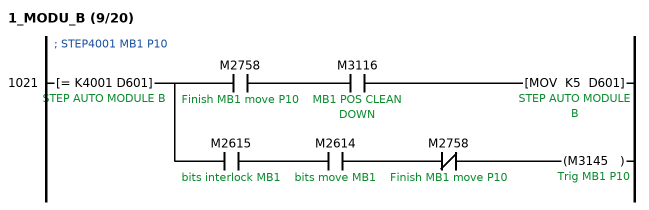
[picture p24: ladder of 1_MODU_B, rungs at steps 1021 to 1021]
; STEP4001 MB1 P10
1021  LD=     K4001 D601  ; STEP AUTO MODULE B
      MPS
      AND     M2758  ; Finish MB1 move P10
      AND     M3116  ; MB1 POS CLEAN DOWN
      MOV     K5 D601
      MPP
      AND     M2615  ; bits interlock MB1
      AND     M2614  ; bits move MB1
      ANI     M2758  ; Finish MB1 move P10
      OUT     M3145  ; Trig MB1 P10
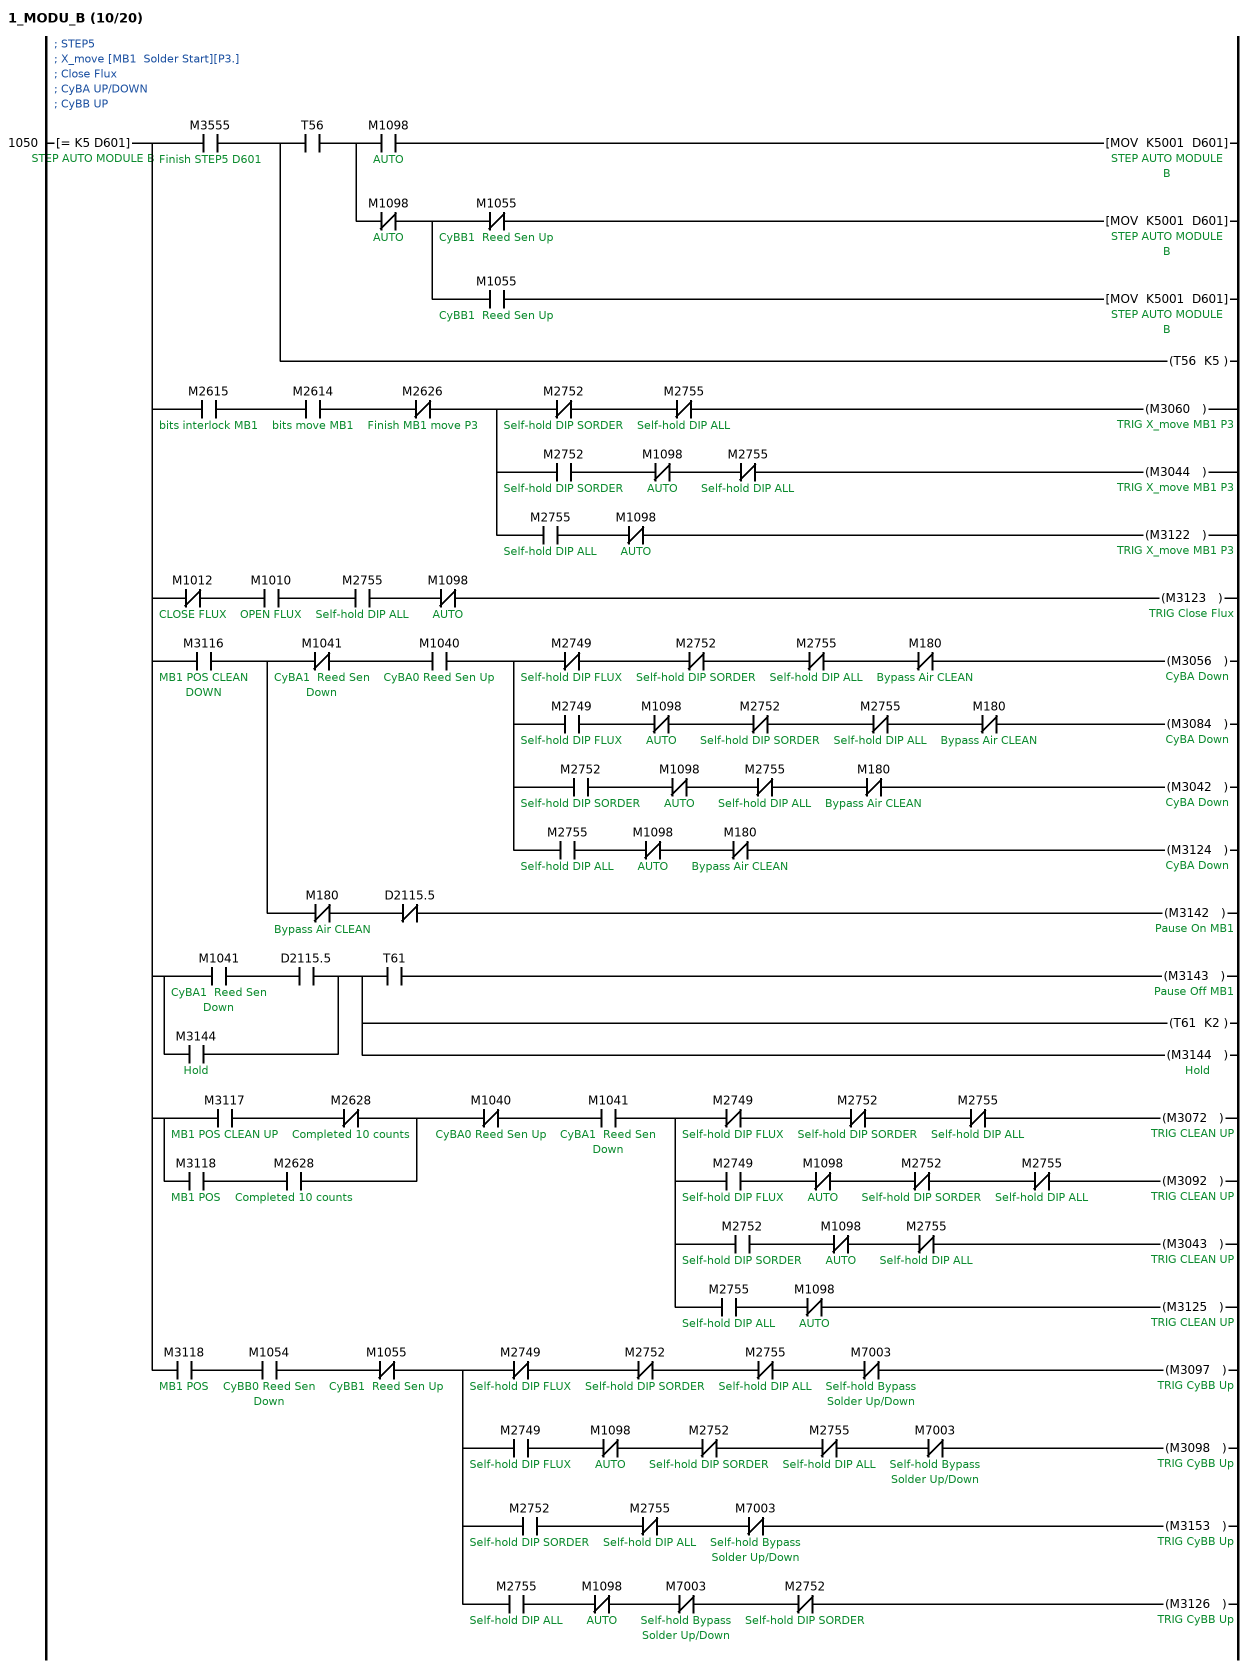
; STEP5
; X_move [MB1  Solder Start][P3.]
; Close Flux
; CyBA UP/DOWN
; CyBB UP
1050  LD=     K5 D601  ; STEP AUTO MODULE B
      MPS
      AND     M3555  ; Finish STEP5 D601
      MPS
      AND     T56
      MPS
      AND     M1098  ; AUTO
      MOV     K5001 D601
      MPP
      ANI     M1098  ; AUTO
      MPS
      ANI     M1055  ; CyBB1  Reed Sen Up
      MOV     K5001 D601
      MPP
      AND     M1055  ; CyBB1  Reed Sen Up
      MOV     K5001 D601
      MPP
      OUT     T56 K5
      MRD
      AND     M2615  ; bits interlock MB1
      AND     M2614  ; bits move MB1
      ANI     M2626  ; Finish MB1 move P3
      MPS
      ANI     M2752  ; Self-hold DIP SORDER
      ANI     M2755  ; Self-hold DIP ALL
      OUT     M3060  ; TRIG X_move MB1 P3
        [note] TRIG X_move MB1 P3
      MRD
      AND     M2752  ; Self-hold DIP SORDER
      ANI     M1098  ; AUTO
      ANI     M2755  ; Self-hold DIP ALL
      OUT     M3044  ; TRIG X_move MB1 P3
      MPP
      AND     M2755  ; Self-hold DIP ALL
      ANI     M1098  ; AUTO
      OUT     M3122  ; TRIG X_move MB1 P3
      MRD
      ANI     M1012  ; CLOSE FLUX
      AND     M1010  ; OPEN FLUX
      AND     M2755  ; Self-hold DIP ALL
      ANI     M1098  ; AUTO
      OUT     M3123  ; TRIG Close Flux
      MRD
      AND     M3116  ; MB1 POS CLEAN DOWN
      MPS
      ANI     M1041  ; CyBA1  Reed Sen Down
      AND     M1040  ; CyBA0 Reed Sen Up
      MPS
      ANI     M2749  ; Self-hold DIP FLUX
      ANI     M2752  ; Self-hold DIP SORDER
      ANI     M2755  ; Self-hold DIP ALL
      ANI     M180  ; Bypass Air CLEAN
      OUT     M3056  ; CyBA Down
        [note] TRIG CLEAN DOWN
      MRD
      AND     M2749  ; Self-hold DIP FLUX
      ANI     M1098  ; AUTO
      ANI     M2752  ; Self-hold DIP SORDER
      ANI     M2755  ; Self-hold DIP ALL
      ANI     M180  ; Bypass Air CLEAN
      OUT     M3084  ; CyBA Down
      MRD
      AND     M2752  ; Self-hold DIP SORDER
      ANI     M1098  ; AUTO
      ANI     M2755  ; Self-hold DIP ALL
      ANI     M180  ; Bypass Air CLEAN
      OUT     M3042  ; CyBA Down
      MPP
      AND     M2755  ; Self-hold DIP ALL
      ANI     M1098  ; AUTO
      ANI     M180  ; Bypass Air CLEAN
      OUT     M3124  ; CyBA Down
      MPP
      ANI     M180  ; Bypass Air CLEAN
      ANI     D2115.5
      OUT     M3142  ; Pause On MB1
      MRD
      LD      M1041  ; CyBA1  Reed Sen Down
      AND     D2115.5
      OR      M3144  ; Hold
      ANB
      MPS
      AND     T61
      OUT     M3143  ; Pause Off MB1
      MPP
      OUT     T61 K2
      OUT     M3144  ; Hold
      MRD
      LD      M3117  ; MB1 POS CLEAN UP
      ANI     M2628  ; Completed 10 counts
      LD      M3118  ; MB1 POS
      AND     M2628  ; Completed 10 counts
      ORB
      ANB
      ANI     M1040  ; CyBA0 Reed Sen Up
      AND     M1041  ; CyBA1  Reed Sen Down
      MPS
      ANI     M2749  ; Self-hold DIP FLUX
      ANI     M2752  ; Self-hold DIP SORDER
      ANI     M2755  ; Self-hold DIP ALL
      OUT     M3072  ; TRIG CLEAN UP
        [note] TRIG CLEAN UP
      MRD
      AND     M2749  ; Self-hold DIP FLUX
      ANI     M1098  ; AUTO
      ANI     M2752  ; Self-hold DIP SORDER
      ANI     M2755  ; Self-hold DIP ALL
      OUT     M3092  ; TRIG CLEAN UP
      MRD
      AND     M2752  ; Self-hold DIP SORDER
      ANI     M1098  ; AUTO
      ANI     M2755  ; Self-hold DIP ALL
      OUT     M3043  ; TRIG CLEAN UP
      MPP
      AND     M2755  ; Self-hold DIP ALL
      ANI     M1098  ; AUTO
      OUT     M3125  ; TRIG CLEAN UP
      MPP
      AND     M3118  ; MB1 POS
      AND     M1054  ; CyBB0 Reed Sen Down
      ANI     M1055  ; CyBB1  Reed Sen Up
      MPS
      ANI     M2749  ; Self-hold DIP FLUX
      ANI     M2752  ; Self-hold DIP SORDER
      ANI     M2755  ; Self-hold DIP ALL
      ANI     M7003  ; Self-hold Bypass Solder Up/Down
      OUT     M3097  ; TRIG CyBB Up
        [note] TRIG CyBB Up
      MRD
      AND     M2749  ; Self-hold DIP FLUX
      ANI     M1098  ; AUTO
      ANI     M2752  ; Self-hold DIP SORDER
      ANI     M2755  ; Self-hold DIP ALL
      ANI     M7003  ; Self-hold Bypass Solder Up/Down
      OUT     M3098  ; TRIG CyBB Up
      MRD
      AND     M2752  ; Self-hold DIP SORDER
      ANI     M2755  ; Self-hold DIP ALL
      ANI     M7003  ; Self-hold Bypass Solder Up/Down
      OUT     M3153  ; TRIG CyBB Up
      MPP
      AND     M2755  ; Self-hold DIP ALL
      ANI     M1098  ; AUTO
      ANI     M7003  ; Self-hold Bypass Solder Up/Down
      ANI     M2752  ; Self-hold DIP SORDER
      OUT     M3126  ; TRIG CyBB Up
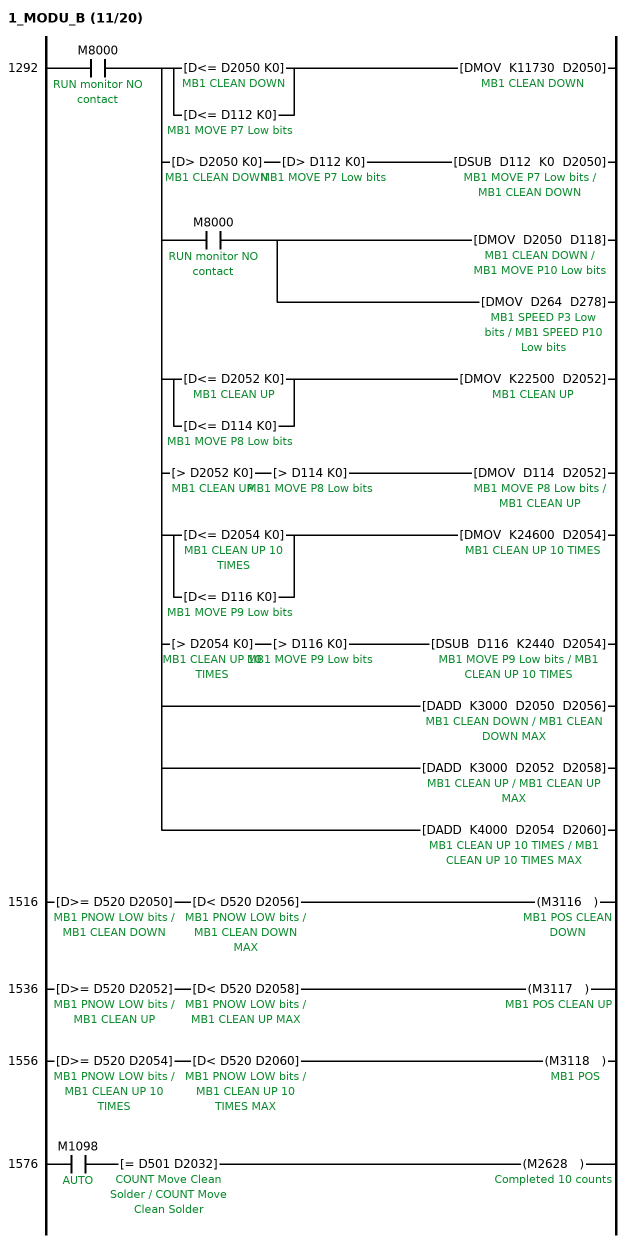
1292  LD      M8000  ; RUN monitor NO contact
      MPS
      LDD<=   D2050 K0  ; MB1 CLEAN DOWN
      ORD<=   D112 K0  ; MB1 MOVE P7 Low bits
      ANB
      DMOV    K11730 D2050
      MRD
      ANDD>   D2050 K0  ; MB1 CLEAN DOWN
      ANDD>   D112 K0  ; MB1 MOVE P7 Low bits
      DSUB    D112 K0 D2050
      MRD
      AND     M8000  ; RUN monitor NO contact
      DMOV    D2050 D118  ; MB1 MOVE P10 Low bits
      DMOV    D264 D278  ; MB1 SPEED P3 Low bits / MB1 SPEED P10 Low bits
      MRD
      LDD<=   D2052 K0  ; MB1 CLEAN UP
      ORD<=   D114 K0  ; MB1 MOVE P8 Low bits
      ANB
      DMOV    K22500 D2052
      MRD
      AND>    D2052 K0  ; MB1 CLEAN UP
      AND>    D114 K0  ; MB1 MOVE P8 Low bits
      DMOV    D114 D2052
      MRD
      LDD<=   D2054 K0  ; MB1 CLEAN UP 10 TIMES
      ORD<=   D116 K0  ; MB1 MOVE P9 Low bits
      ANB
      DMOV    K24600 D2054
      MRD
      AND>    D2054 K0  ; MB1 CLEAN UP 10 TIMES
      AND>    D116 K0  ; MB1 MOVE P9 Low bits
      DSUB    D116 K2440 D2054
      MPP
      DADD    K3000 D2050 D2056  ; MB1 CLEAN DOWN MAX
      DADD    K3000 D2052 D2058  ; MB1 CLEAN UP MAX
      DADD    K4000 D2054 D2060  ; MB1 CLEAN UP 10 TIMES MAX
1516  LDD>=   D520 D2050  ; MB1 PNOW LOW bits / MB1 CLEAN DOWN
      ANDD<   D520 D2056  ; MB1 PNOW LOW bits / MB1 CLEAN DOWN MAX
      OUT     M3116  ; MB1 POS CLEAN DOWN
1536  LDD>=   D520 D2052  ; MB1 PNOW LOW bits / MB1 CLEAN UP
      ANDD<   D520 D2058  ; MB1 PNOW LOW bits / MB1 CLEAN UP MAX
      OUT     M3117  ; MB1 POS CLEAN UP
1556  LDD>=   D520 D2054  ; MB1 PNOW LOW bits / MB1 CLEAN UP 10 TIMES
      ANDD<   D520 D2060  ; MB1 PNOW LOW bits / MB1 CLEAN UP 10 TIMES MAX
      OUT     M3118  ; MB1 POS
1576  LD      M1098  ; AUTO
      AND=    D501 D2032  ; COUNT Move Clean Solder / COUNT Move Clean Solder
      OUT     M2628  ; Completed 10 counts
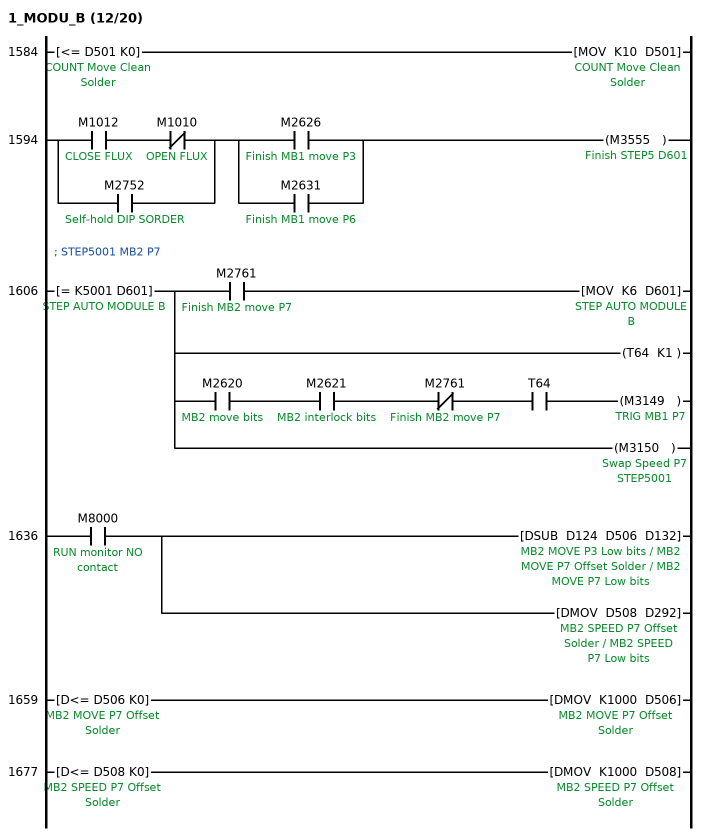
1584  LD<=    D501 K0  ; COUNT Move Clean Solder
      MOV     K10 D501
1594  LD      M1012  ; CLOSE FLUX
      ANI     M1010  ; OPEN FLUX
      OR      M2752  ; Self-hold DIP SORDER
      LD      M2626  ; Finish MB1 move P3
      OR      M2631  ; Finish MB1 move P6
      ANB
      OUT     M3555  ; Finish STEP5 D601
; STEP5001 MB2 P7
1606  LD=     K5001 D601  ; STEP AUTO MODULE B
      MPS
      AND     M2761  ; Finish MB2 move P7
      MOV     K6 D601
      MPP
      OUT     T64 K1
      MPS
      AND     M2620  ; MB2 move bits
      AND     M2621  ; MB2 interlock bits
      ANI     M2761  ; Finish MB2 move P7
      AND     T64
      OUT     M3149  ; TRIG MB1 P7
      MPP
      OUT     M3150  ; Swap Speed P7 STEP5001
1636  LD      M8000  ; RUN monitor NO contact
      DSUB    D124 D506 D132  ; MB2 MOVE P3 Low bits / MB2 MOVE P7 Offset Solder / MB2 MOVE P7 Low bits
      DMOV    D508 D292  ; MB2 SPEED P7 Offset Solder / MB2 SPEED P7 Low bits
1659  LDD<=   D506 K0  ; MB2 MOVE P7 Offset Solder
      DMOV    K1000 D506
1677  LDD<=   D508 K0  ; MB2 SPEED P7 Offset Solder
      DMOV    K1000 D508
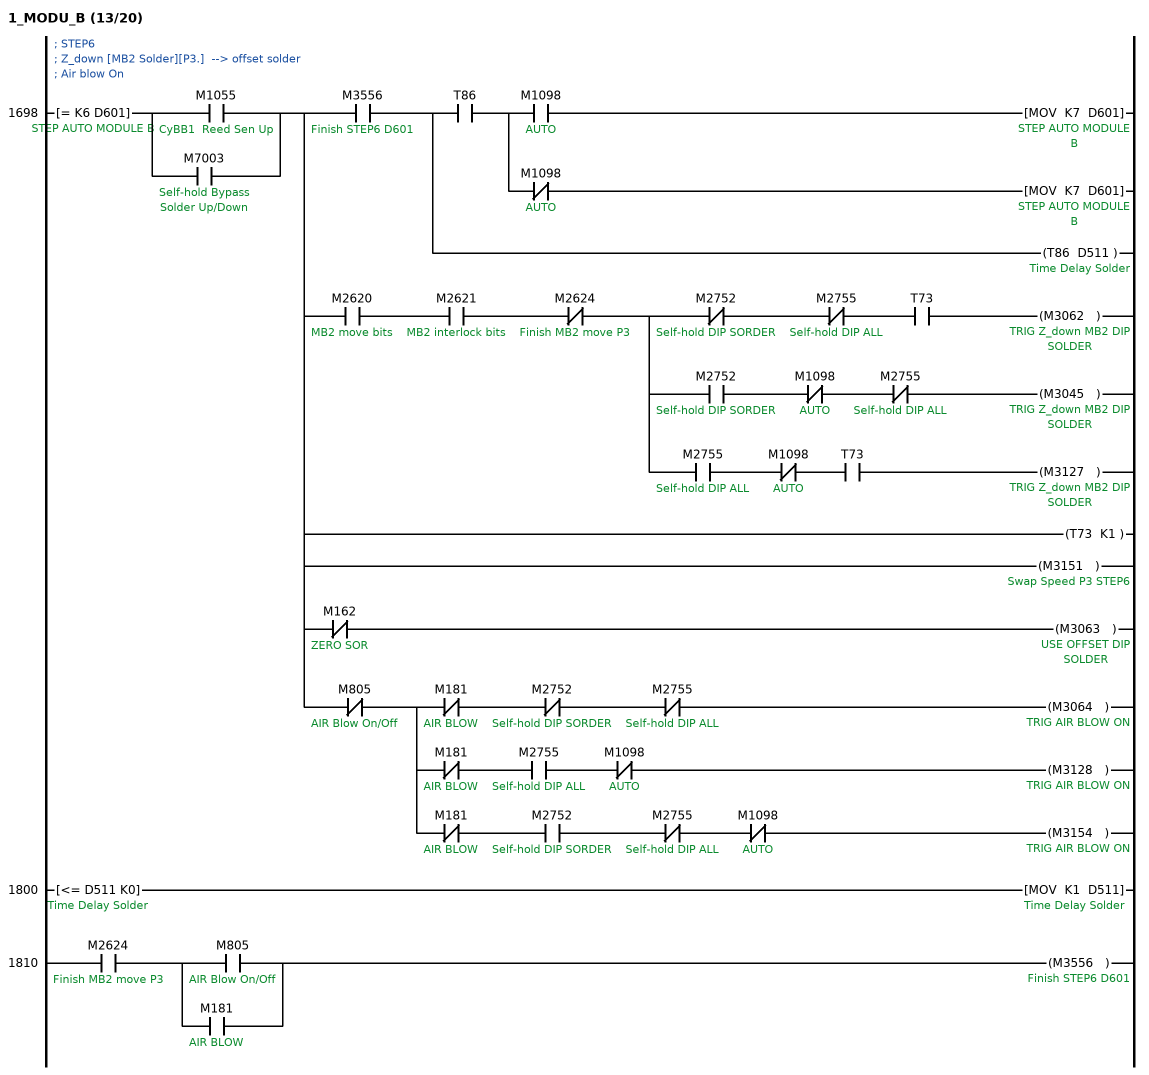
; STEP6
; Z_down [MB2 Solder][P3.]  --> offset solder
; Air blow On
1698  LD=     K6 D601  ; STEP AUTO MODULE B
      LD      M1055  ; CyBB1  Reed Sen Up
      OR      M7003  ; Self-hold Bypass Solder Up/Down
      ANB
      MPS
      AND     M3556  ; Finish STEP6 D601
      MPS
      AND     T86
      MPS
      AND     M1098  ; AUTO
      MOV     K7 D601
      MPP
      ANI     M1098  ; AUTO
      MOV     K7 D601
      MPP
      OUT     T86 D511  ; Time Delay Solder
      MRD
      AND     M2620  ; MB2 move bits
      AND     M2621  ; MB2 interlock bits
      ANI     M2624  ; Finish MB2 move P3
      MPS
      ANI     M2752  ; Self-hold DIP SORDER
      ANI     M2755  ; Self-hold DIP ALL
      AND     T73
      OUT     M3062  ; TRIG Z_down MB2 DIP SOLDER
        [note] TRIG Z_down MB2 DIP SOLDER
      MRD
      AND     M2752  ; Self-hold DIP SORDER
      ANI     M1098  ; AUTO
      ANI     M2755  ; Self-hold DIP ALL
      OUT     M3045  ; TRIG Z_down MB2 DIP SOLDER
      MPP
      AND     M2755  ; Self-hold DIP ALL
      ANI     M1098  ; AUTO
      AND     T73
      OUT     M3127  ; TRIG Z_down MB2 DIP SOLDER
      MPP
      OUT     T73 K1
      OUT     M3151  ; Swap Speed P3 STEP6
      MPS
      ANI     M162  ; ZERO SOR
      OUT     M3063  ; USE OFFSET DIP SOLDER
        [note] USE OFFSET DIP SOLDER
      MPP
      ANI     M805  ; AIR Blow On/Off
      MPS
      ANI     M181  ; AIR BLOW
      ANI     M2752  ; Self-hold DIP SORDER
      ANI     M2755  ; Self-hold DIP ALL
      OUT     M3064  ; TRIG AIR BLOW ON
        [note] TRIG AIR BLOW ON
      MRD
      ANI     M181  ; AIR BLOW
      AND     M2755  ; Self-hold DIP ALL
      ANI     M1098  ; AUTO
      OUT     M3128  ; TRIG AIR BLOW ON
      MPP
      ANI     M181  ; AIR BLOW
      AND     M2752  ; Self-hold DIP SORDER
      ANI     M2755  ; Self-hold DIP ALL
      ANI     M1098  ; AUTO
      OUT     M3154  ; TRIG AIR BLOW ON
1800  LD<=    D511 K0  ; Time Delay Solder
      MOV     K1 D511
1810  LD      M2624  ; Finish MB2 move P3
      LD      M805  ; AIR Blow On/Off
      OR      M181  ; AIR BLOW
      ANB
      OUT     M3556  ; Finish STEP6 D601
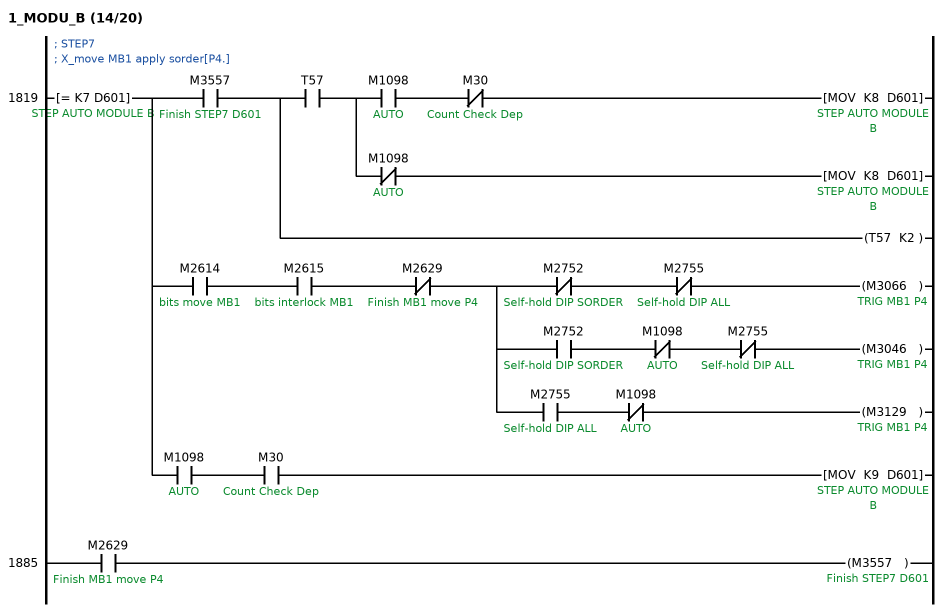
; STEP7
; X_move MB1 apply sorder[P4.]
1819  LD=     K7 D601  ; STEP AUTO MODULE B
      MPS
      AND     M3557  ; Finish STEP7 D601
      MPS
      AND     T57
      MPS
      AND     M1098  ; AUTO
      ANI     M30  ; Count Check Dep
      MOV     K8 D601
      MPP
      ANI     M1098  ; AUTO
      MOV     K8 D601
      MPP
      OUT     T57 K2
      MRD
      AND     M2614  ; bits move MB1
      AND     M2615  ; bits interlock MB1
      ANI     M2629  ; Finish MB1 move P4
      MPS
      ANI     M2752  ; Self-hold DIP SORDER
      ANI     M2755  ; Self-hold DIP ALL
      OUT     M3066  ; TRIG MB1 P4
        [note] TRIG MB1 P4
      MRD
      AND     M2752  ; Self-hold DIP SORDER
      ANI     M1098  ; AUTO
      ANI     M2755  ; Self-hold DIP ALL
      OUT     M3046  ; TRIG MB1 P4
      MPP
      AND     M2755  ; Self-hold DIP ALL
      ANI     M1098  ; AUTO
      OUT     M3129  ; TRIG MB1 P4
      MPP
      AND     M1098  ; AUTO
      AND     M30  ; Count Check Dep
      MOV     K9 D601
1885  LD      M2629  ; Finish MB1 move P4
      OUT     M3557  ; Finish STEP7 D601
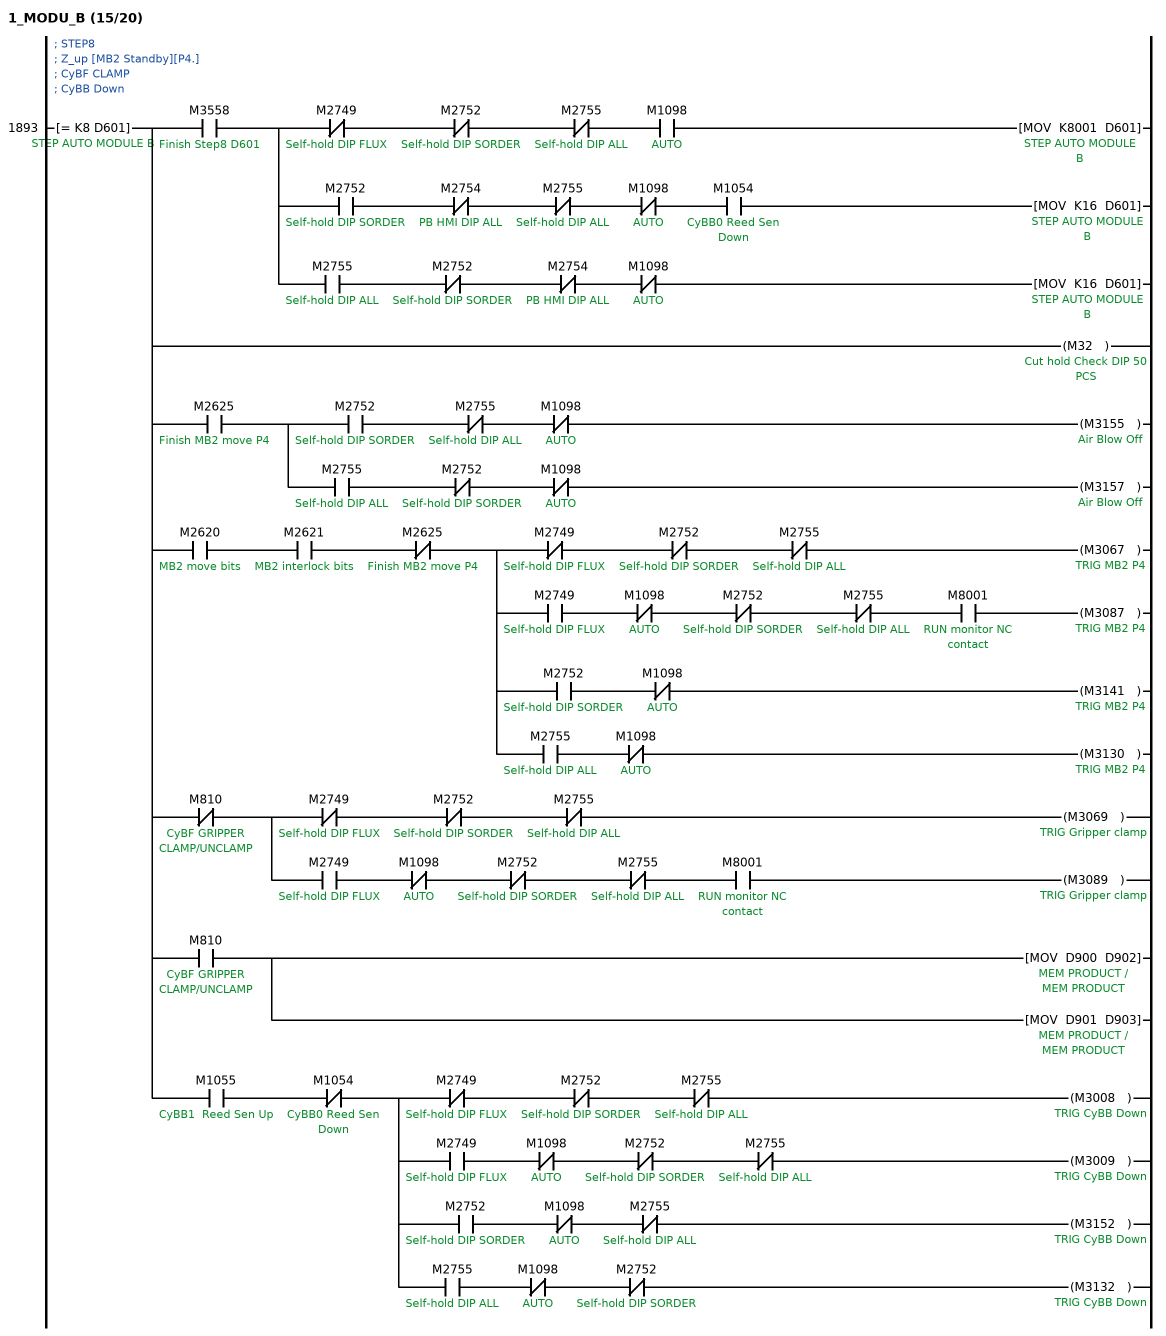
; STEP8
; Z_up [MB2 Standby][P4.]
; CyBF CLAMP
; CyBB Down
1893  LD=     K8 D601  ; STEP AUTO MODULE B
      MPS
      AND     M3558  ; Finish Step8 D601
      MPS
      ANI     M2749  ; Self-hold DIP FLUX
      ANI     M2752  ; Self-hold DIP SORDER
      ANI     M2755  ; Self-hold DIP ALL
      AND     M1098  ; AUTO
      MOV     K8001 D601
      MRD
      AND     M2752  ; Self-hold DIP SORDER
      ANI     M2754  ; PB HMI DIP ALL
      ANI     M2755  ; Self-hold DIP ALL
      ANI     M1098  ; AUTO
      AND     M1054  ; CyBB0 Reed Sen Down
      MOV     K16 D601
      MPP
      AND     M2755  ; Self-hold DIP ALL
      ANI     M2752  ; Self-hold DIP SORDER
      ANI     M2754  ; PB HMI DIP ALL
      ANI     M1098  ; AUTO
      MOV     K16 D601
      MPP
      OUT     M32  ; Cut hold Check DIP 50 PCS
      MPS
      AND     M2625  ; Finish MB2 move P4
      MPS
      AND     M2752  ; Self-hold DIP SORDER
      ANI     M2755  ; Self-hold DIP ALL
      ANI     M1098  ; AUTO
      OUT     M3155  ; Air Blow Off
      MPP
      AND     M2755  ; Self-hold DIP ALL
      ANI     M2752  ; Self-hold DIP SORDER
      ANI     M1098  ; AUTO
      OUT     M3157  ; Air Blow Off
      MRD
      AND     M2620  ; MB2 move bits
      AND     M2621  ; MB2 interlock bits
      ANI     M2625  ; Finish MB2 move P4
      MPS
      ANI     M2749  ; Self-hold DIP FLUX
      ANI     M2752  ; Self-hold DIP SORDER
      ANI     M2755  ; Self-hold DIP ALL
      OUT     M3067  ; TRIG MB2 P4
        [note] TRIG MB2 P4
      MRD
      AND     M2749  ; Self-hold DIP FLUX
      ANI     M1098  ; AUTO
      ANI     M2752  ; Self-hold DIP SORDER
      ANI     M2755  ; Self-hold DIP ALL
      AND     M8001  ; RUN monitor NC contact
      OUT     M3087  ; TRIG MB2 P4
      MRD
      AND     M2752  ; Self-hold DIP SORDER
      ANI     M1098  ; AUTO
      OUT     M3141  ; TRIG MB2 P4
      MPP
      AND     M2755  ; Self-hold DIP ALL
      ANI     M1098  ; AUTO
      OUT     M3130  ; TRIG MB2 P4
      MRD
      ANI     M810  ; CyBF GRIPPER CLAMP/UNCLAMP
      MPS
      ANI     M2749  ; Self-hold DIP FLUX
      ANI     M2752  ; Self-hold DIP SORDER
      ANI     M2755  ; Self-hold DIP ALL
      OUT     M3069  ; TRIG Gripper clamp
        [note] TRIG Gripper clamp
      MPP
      AND     M2749  ; Self-hold DIP FLUX
      ANI     M1098  ; AUTO
      ANI     M2752  ; Self-hold DIP SORDER
      ANI     M2755  ; Self-hold DIP ALL
      AND     M8001  ; RUN monitor NC contact
      OUT     M3089  ; TRIG Gripper clamp
      MRD
      AND     M810  ; CyBF GRIPPER CLAMP/UNCLAMP
      MOV     D900 D902
      MOV     D901 D903
      MPP
      AND     M1055  ; CyBB1  Reed Sen Up
      ANI     M1054  ; CyBB0 Reed Sen Down
      MPS
      ANI     M2749  ; Self-hold DIP FLUX
      ANI     M2752  ; Self-hold DIP SORDER
      ANI     M2755  ; Self-hold DIP ALL
      OUT     M3008  ; TRIG CyBB Down
        [note] TRIG CyBB Down
      MRD
      AND     M2749  ; Self-hold DIP FLUX
      ANI     M1098  ; AUTO
      ANI     M2752  ; Self-hold DIP SORDER
      ANI     M2755  ; Self-hold DIP ALL
      OUT     M3009  ; TRIG CyBB Down
      MRD
      AND     M2752  ; Self-hold DIP SORDER
      ANI     M1098  ; AUTO
      ANI     M2755  ; Self-hold DIP ALL
      OUT     M3152  ; TRIG CyBB Down
      MPP
      AND     M2755  ; Self-hold DIP ALL
      ANI     M1098  ; AUTO
      ANI     M2752  ; Self-hold DIP SORDER
      OUT     M3132  ; TRIG CyBB Down
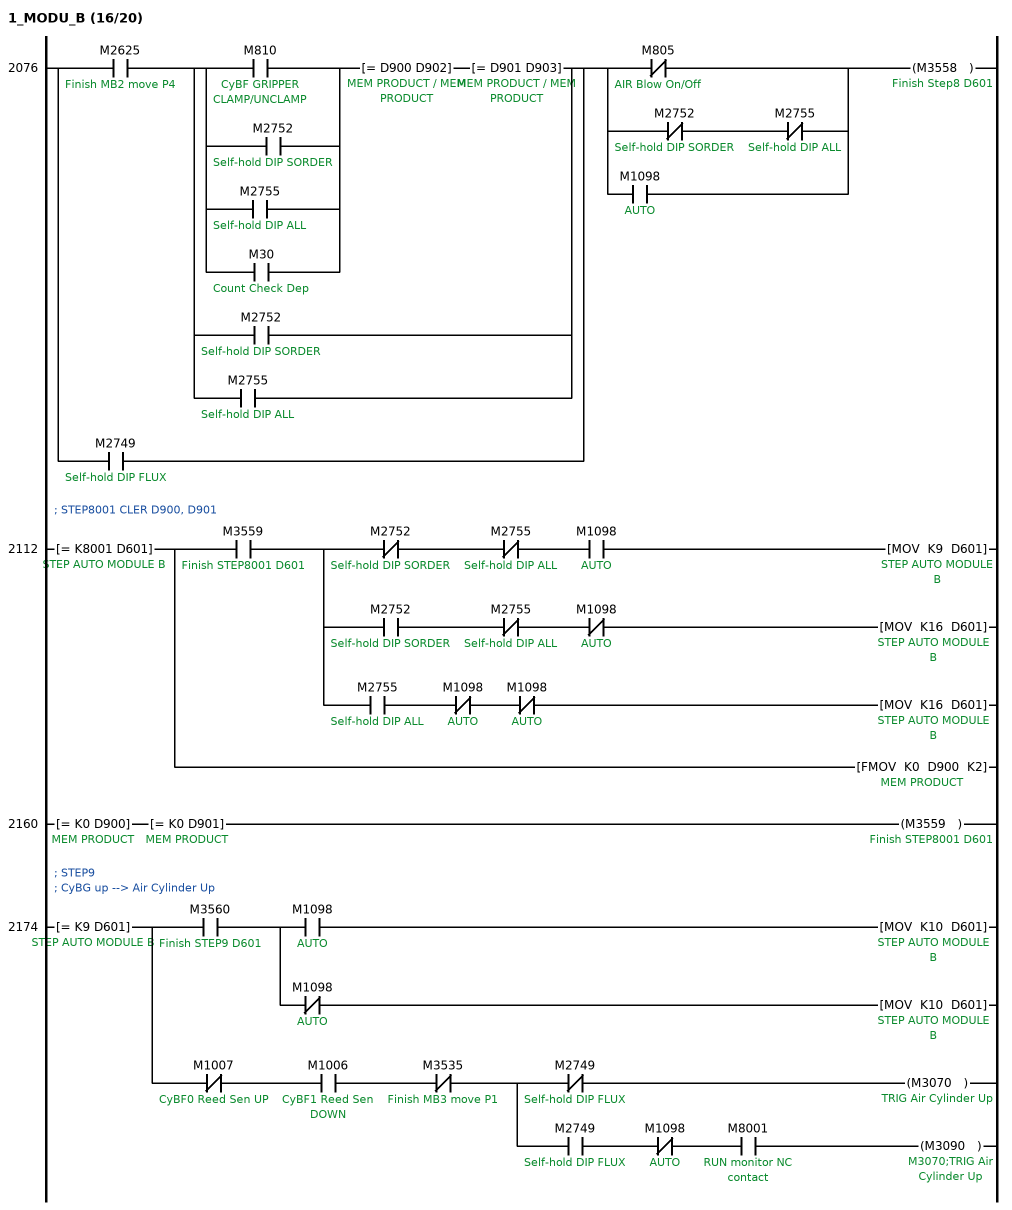
2076  LD      M2625  ; Finish MB2 move P4
      LD      M810  ; CyBF GRIPPER CLAMP/UNCLAMP
      OR      M2752  ; Self-hold DIP SORDER
      OR      M2755  ; Self-hold DIP ALL
      OR      M30  ; Count Check Dep
      AND=    D900 D902  ; MEM PRODUCT / MEM PRODUCT
      AND=    D901 D903  ; MEM PRODUCT / MEM PRODUCT
      OR      M2752  ; Self-hold DIP SORDER
      OR      M2755  ; Self-hold DIP ALL
      ANB
      OR      M2749  ; Self-hold DIP FLUX
      LDI     M805  ; AIR Blow On/Off
      LDI     M2752  ; Self-hold DIP SORDER
      ANI     M2755  ; Self-hold DIP ALL
      ORB
      OR      M1098  ; AUTO
      ANB
      OUT     M3558  ; Finish Step8 D601
; STEP8001 CLER D900, D901
2112  LD=     K8001 D601  ; STEP AUTO MODULE B
      MPS
      AND     M3559  ; Finish STEP8001 D601
      MPS
      ANI     M2752  ; Self-hold DIP SORDER
      ANI     M2755  ; Self-hold DIP ALL
      AND     M1098  ; AUTO
      MOV     K9 D601
      MRD
      AND     M2752  ; Self-hold DIP SORDER
      ANI     M2755  ; Self-hold DIP ALL
      ANI     M1098  ; AUTO
      MOV     K16 D601
      MPP
      AND     M2755  ; Self-hold DIP ALL
      ANI     M1098  ; AUTO
      ANI     M1098  ; AUTO
      MOV     K16 D601
      MPP
      FMOV    K0 D900 K2
2160  LD=     K0 D900  ; MEM PRODUCT
      AND=    K0 D901  ; MEM PRODUCT
      OUT     M3559  ; Finish STEP8001 D601
; STEP9
; CyBG up --> Air Cylinder Up
2174  LD=     K9 D601  ; STEP AUTO MODULE B
      MPS
      AND     M3560  ; Finish STEP9 D601
      MPS
      AND     M1098  ; AUTO
      MOV     K10 D601
      MPP
      ANI     M1098  ; AUTO
      MOV     K10 D601
      MPP
      ANI     M1007  ; CyBF0 Reed Sen UP
      AND     M1006  ; CyBF1 Reed Sen DOWN
      ANI     M3535  ; Finish MB3 move P1
      MPS
      ANI     M2749  ; Self-hold DIP FLUX
      OUT     M3070  ; TRIG Air Cylinder Up
        [note] TRIG Air Cylinder Up
      MPP
      AND     M2749  ; Self-hold DIP FLUX
      ANI     M1098  ; AUTO
      AND     M8001  ; RUN monitor NC contact
      OUT     M3090  ; M3070;TRIG Air Cylinder Up
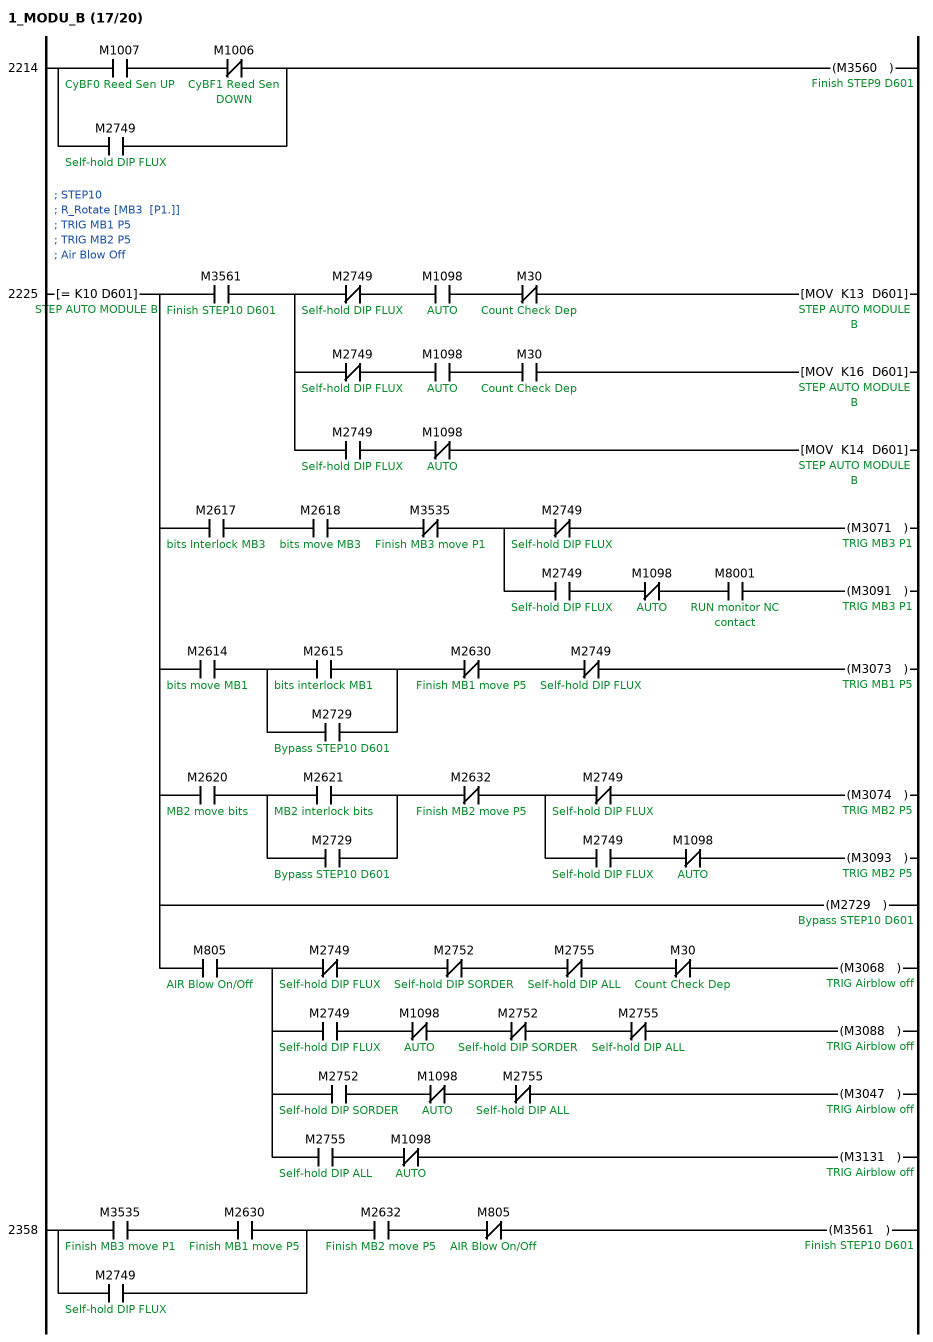
2214  LD      M1007  ; CyBF0 Reed Sen UP
      ANI     M1006  ; CyBF1 Reed Sen DOWN
      OR      M2749  ; Self-hold DIP FLUX
      OUT     M3560  ; Finish STEP9 D601
; STEP10
; R_Rotate [MB3  [P1.]]
; TRIG MB1 P5
; TRIG MB2 P5
; Air Blow Off
2225  LD=     K10 D601  ; STEP AUTO MODULE B
      MPS
      AND     M3561  ; Finish STEP10 D601
      MPS
      ANI     M2749  ; Self-hold DIP FLUX
      AND     M1098  ; AUTO
      ANI     M30  ; Count Check Dep
      MOV     K13 D601
      MRD
      ANI     M2749  ; Self-hold DIP FLUX
      AND     M1098  ; AUTO
      AND     M30  ; Count Check Dep
      MOV     K16 D601
      MPP
      AND     M2749  ; Self-hold DIP FLUX
      ANI     M1098  ; AUTO
      MOV     K14 D601
      MRD
      AND     M2617  ; bits Interlock MB3
      AND     M2618  ; bits move MB3
      ANI     M3535  ; Finish MB3 move P1
      MPS
      ANI     M2749  ; Self-hold DIP FLUX
      OUT     M3071  ; TRIG MB3 P1
        [note] TRIG MB3 P1
      MPP
      AND     M2749  ; Self-hold DIP FLUX
      ANI     M1098  ; AUTO
      AND     M8001  ; RUN monitor NC contact
      OUT     M3091  ; TRIG MB3 P1
      MRD
      AND     M2614  ; bits move MB1
      LD      M2615  ; bits interlock MB1
      OR      M2729  ; Bypass STEP10 D601
      ANB
      ANI     M2630  ; Finish MB1 move P5
      ANI     M2749  ; Self-hold DIP FLUX
      OUT     M3073  ; TRIG MB1 P5
        [note] TRIG MB1 P5
      MRD
      AND     M2620  ; MB2 move bits
      LD      M2621  ; MB2 interlock bits
      OR      M2729  ; Bypass STEP10 D601
      ANB
      ANI     M2632  ; Finish MB2 move P5
      MPS
      ANI     M2749  ; Self-hold DIP FLUX
      OUT     M3074  ; TRIG MB2 P5
        [note] TRIG MB2 P5
      MPP
      AND     M2749  ; Self-hold DIP FLUX
      ANI     M1098  ; AUTO
      OUT     M3093  ; TRIG MB2 P5
      MPP
      OUT     M2729  ; Bypass STEP10 D601
      AND     M805  ; AIR Blow On/Off
      MPS
      ANI     M2749  ; Self-hold DIP FLUX
      ANI     M2752  ; Self-hold DIP SORDER
      ANI     M2755  ; Self-hold DIP ALL
      ANI     M30  ; Count Check Dep
      OUT     M3068  ; TRIG Airblow off
        [note] TRIG Airblow off
      MRD
      AND     M2749  ; Self-hold DIP FLUX
      ANI     M1098  ; AUTO
      ANI     M2752  ; Self-hold DIP SORDER
      ANI     M2755  ; Self-hold DIP ALL
      OUT     M3088  ; TRIG Airblow off
      MRD
      AND     M2752  ; Self-hold DIP SORDER
      ANI     M1098  ; AUTO
      ANI     M2755  ; Self-hold DIP ALL
      OUT     M3047  ; TRIG Airblow off
      MPP
      AND     M2755  ; Self-hold DIP ALL
      ANI     M1098  ; AUTO
      OUT     M3131  ; TRIG Airblow off
2358  LD      M3535  ; Finish MB3 move P1
      AND     M2630  ; Finish MB1 move P5
      OR      M2749  ; Self-hold DIP FLUX
      AND     M2632  ; Finish MB2 move P5
      ANI     M805  ; AIR Blow On/Off
      OUT     M3561  ; Finish STEP10 D601
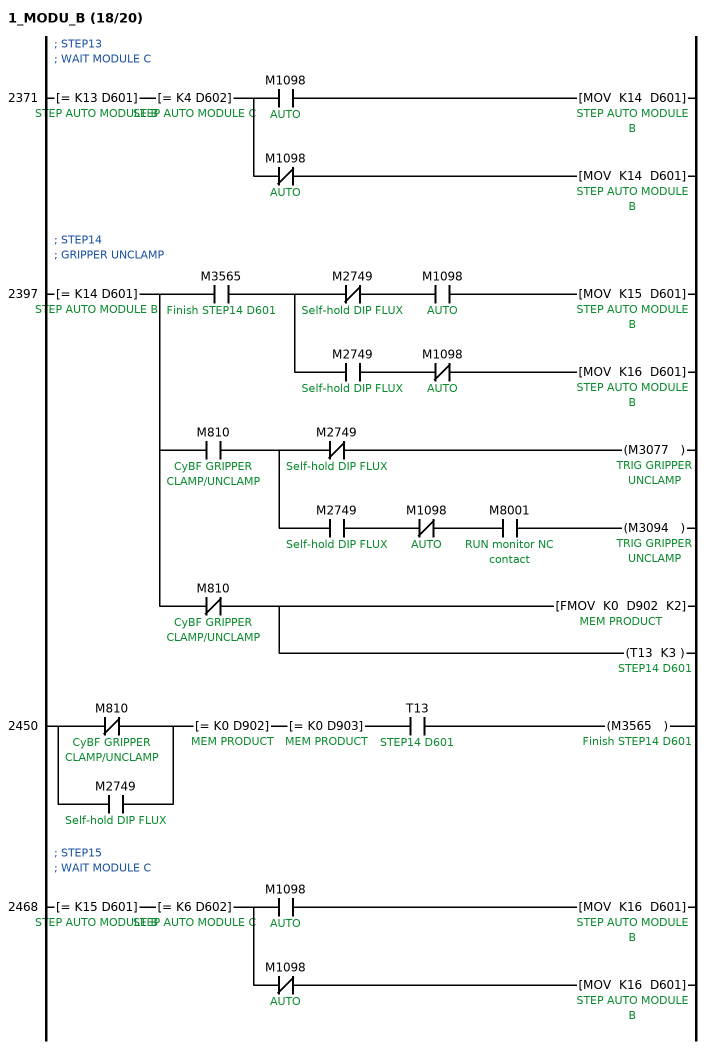
; STEP13
; WAIT MODULE C
2371  LD=     K13 D601  ; STEP AUTO MODULE B
      AND=    K4 D602  ; STEP AUTO MODULE C
      MPS
      AND     M1098  ; AUTO
      MOV     K14 D601
      MPP
      ANI     M1098  ; AUTO
      MOV     K14 D601
; STEP14
; GRIPPER UNCLAMP
2397  LD=     K14 D601  ; STEP AUTO MODULE B
      MPS
      AND     M3565  ; Finish STEP14 D601
      MPS
      ANI     M2749  ; Self-hold DIP FLUX
      AND     M1098  ; AUTO
      MOV     K15 D601
      MPP
      AND     M2749  ; Self-hold DIP FLUX
      ANI     M1098  ; AUTO
      MOV     K16 D601
      MRD
      AND     M810  ; CyBF GRIPPER CLAMP/UNCLAMP
      MPS
      ANI     M2749  ; Self-hold DIP FLUX
      OUT     M3077  ; TRIG GRIPPER UNCLAMP
        [note] TRIG GRIPPER UNCLAMP
      MPP
      AND     M2749  ; Self-hold DIP FLUX
      ANI     M1098  ; AUTO
      AND     M8001  ; RUN monitor NC contact
      OUT     M3094  ; TRIG GRIPPER UNCLAMP
      MPP
      ANI     M810  ; CyBF GRIPPER CLAMP/UNCLAMP
      FMOV    K0 D902 K2
      OUT     T13 K3  ; STEP14 D601
2450  LDI     M810  ; CyBF GRIPPER CLAMP/UNCLAMP
      OR      M2749  ; Self-hold DIP FLUX
      AND=    K0 D902  ; MEM PRODUCT
      AND=    K0 D903  ; MEM PRODUCT
      AND     T13  ; STEP14 D601
      OUT     M3565  ; Finish STEP14 D601
; STEP15
; WAIT MODULE C
2468  LD=     K15 D601  ; STEP AUTO MODULE B
      AND=    K6 D602  ; STEP AUTO MODULE C
      MPS
      AND     M1098  ; AUTO
      MOV     K16 D601
      MPP
      ANI     M1098  ; AUTO
      MOV     K16 D601
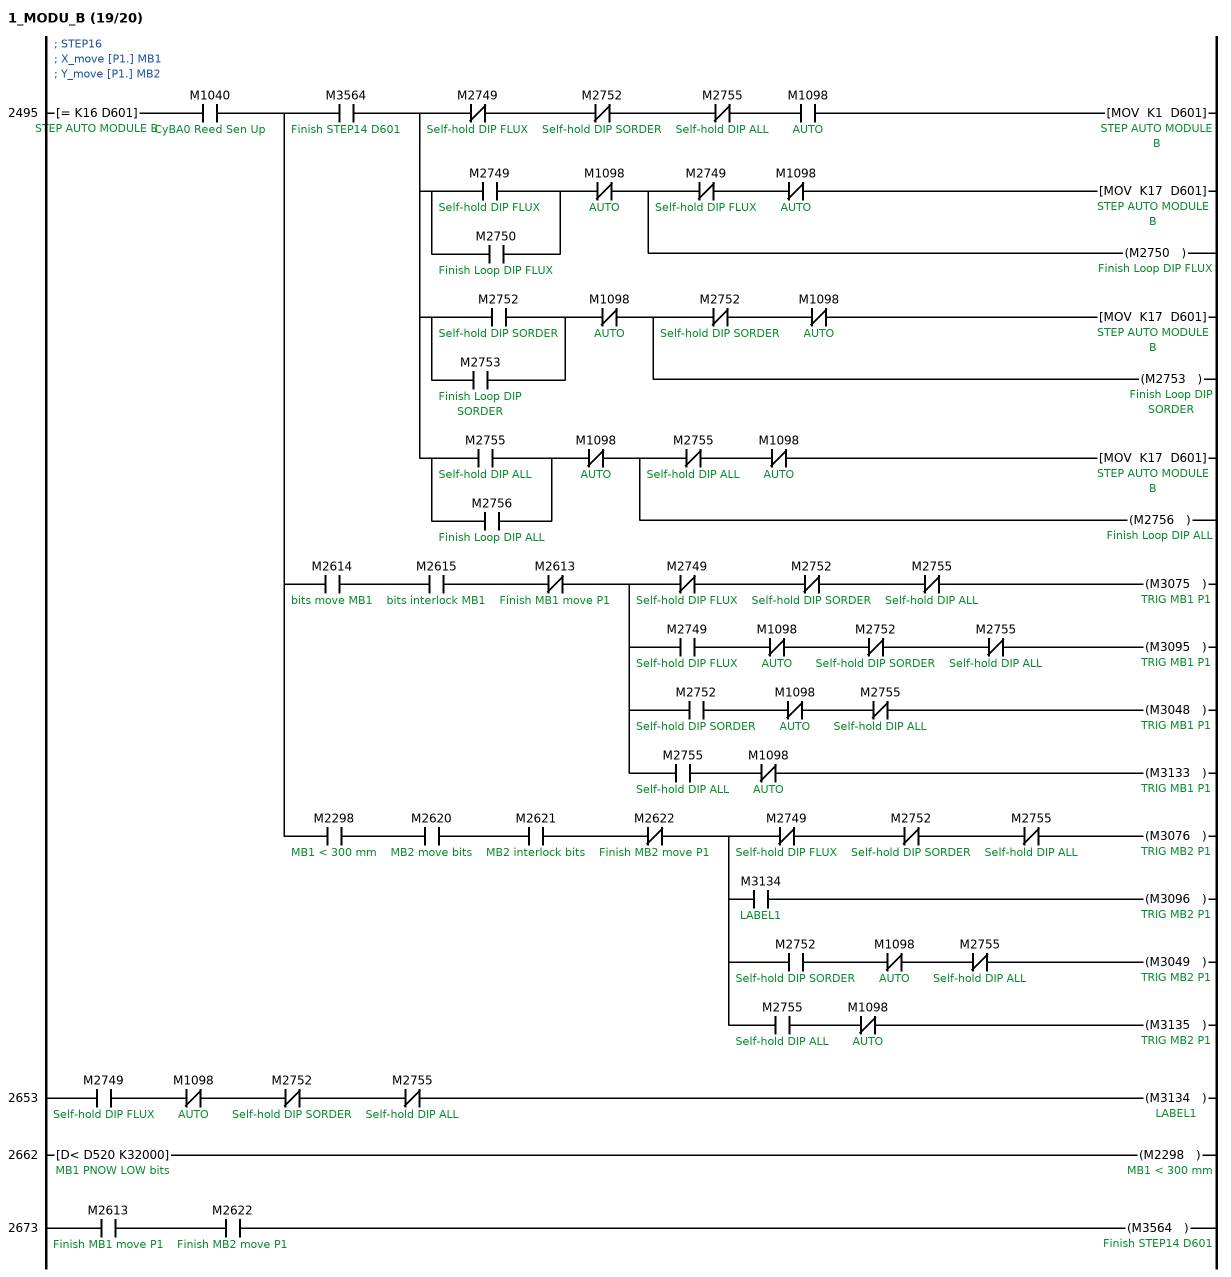
; STEP16
; X_move [P1.] MB1
; Y_move [P1.] MB2
2495  LD=     K16 D601  ; STEP AUTO MODULE B
      AND     M1040  ; CyBA0 Reed Sen Up
      MPS
      AND     M3564  ; Finish STEP14 D601
      MPS
      ANI     M2749  ; Self-hold DIP FLUX
      ANI     M2752  ; Self-hold DIP SORDER
      ANI     M2755  ; Self-hold DIP ALL
      AND     M1098  ; AUTO
      MOV     K1 D601
      MRD
      LD      M2749  ; Self-hold DIP FLUX
      OR      M2750  ; Finish Loop DIP FLUX
      ANB
      ANI     M1098  ; AUTO
      MPS
      ANI     M2749  ; Self-hold DIP FLUX
      ANI     M1098  ; AUTO
      MOV     K17 D601
      MPP
      OUT     M2750  ; Finish Loop DIP FLUX
      MRD
      LD      M2752  ; Self-hold DIP SORDER
      OR      M2753  ; Finish Loop DIP SORDER
      ANB
      ANI     M1098  ; AUTO
      MPS
      ANI     M2752  ; Self-hold DIP SORDER
      ANI     M1098  ; AUTO
      MOV     K17 D601
      MPP
      OUT     M2753  ; Finish Loop DIP SORDER
      MPP
      LD      M2755  ; Self-hold DIP ALL
      OR      M2756  ; Finish Loop DIP ALL
      ANB
      ANI     M1098  ; AUTO
      MPS
      ANI     M2755  ; Self-hold DIP ALL
      ANI     M1098  ; AUTO
      MOV     K17 D601
      MPP
      OUT     M2756  ; Finish Loop DIP ALL
      MRD
      AND     M2614  ; bits move MB1
      AND     M2615  ; bits interlock MB1
      ANI     M2613  ; Finish MB1 move P1
      MPS
      ANI     M2749  ; Self-hold DIP FLUX
      ANI     M2752  ; Self-hold DIP SORDER
      ANI     M2755  ; Self-hold DIP ALL
      OUT     M3075  ; TRIG MB1 P1
        [note] TRIG MB1 P1
      MRD
      AND     M2749  ; Self-hold DIP FLUX
      ANI     M1098  ; AUTO
      ANI     M2752  ; Self-hold DIP SORDER
      ANI     M2755  ; Self-hold DIP ALL
      OUT     M3095  ; TRIG MB1 P1
      MRD
      AND     M2752  ; Self-hold DIP SORDER
      ANI     M1098  ; AUTO
      ANI     M2755  ; Self-hold DIP ALL
      OUT     M3048  ; TRIG MB1 P1
      MPP
      AND     M2755  ; Self-hold DIP ALL
      ANI     M1098  ; AUTO
      OUT     M3133  ; TRIG MB1 P1
      MPP
      AND     M2298  ; MB1 < 300 mm
      AND     M2620  ; MB2 move bits
      AND     M2621  ; MB2 interlock bits
      ANI     M2622  ; Finish MB2 move P1
      MPS
      ANI     M2749  ; Self-hold DIP FLUX
      ANI     M2752  ; Self-hold DIP SORDER
      ANI     M2755  ; Self-hold DIP ALL
      OUT     M3076  ; TRIG MB2 P1
        [note] TRIG MB2 P1
      MRD
      AND     M3134  ; LABEL1
      OUT     M3096  ; TRIG MB2 P1
      MRD
      AND     M2752  ; Self-hold DIP SORDER
      ANI     M1098  ; AUTO
      ANI     M2755  ; Self-hold DIP ALL
      OUT     M3049  ; TRIG MB2 P1
      MPP
      AND     M2755  ; Self-hold DIP ALL
      ANI     M1098  ; AUTO
      OUT     M3135  ; TRIG MB2 P1
2653  LD      M2749  ; Self-hold DIP FLUX
      ANI     M1098  ; AUTO
      ANI     M2752  ; Self-hold DIP SORDER
      ANI     M2755  ; Self-hold DIP ALL
      OUT     M3134  ; LABEL1
2662  LDD<    D520 K32000  ; MB1 PNOW LOW bits
      OUT     M2298  ; MB1 < 300 mm
2673  LD      M2613  ; Finish MB1 move P1
      AND     M2622  ; Finish MB2 move P1
      OUT     M3564  ; Finish STEP14 D601
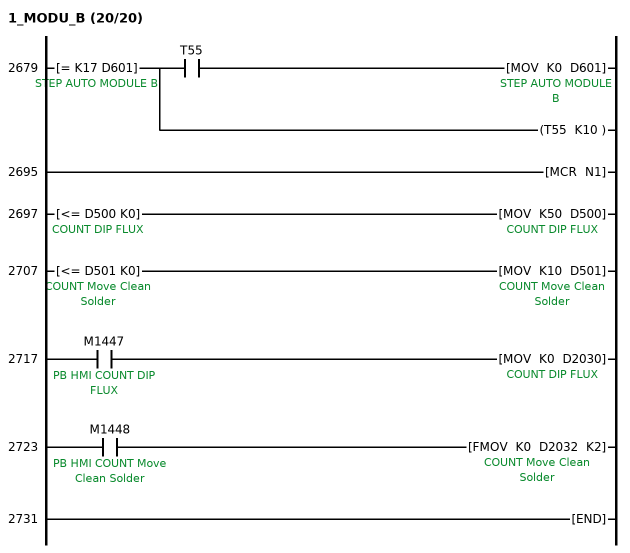
2679  LD=     K17 D601  ; STEP AUTO MODULE B
      MPS
      AND     T55
      MOV     K0 D601
      MPP
      OUT     T55 K10
2695  MCR     N1
2697  LD<=    D500 K0  ; COUNT DIP FLUX
      MOV     K50 D500
2707  LD<=    D501 K0  ; COUNT Move Clean Solder
      MOV     K10 D501
2717  LD      M1447  ; PB HMI COUNT DIP FLUX
      MOV     K0 D2030
2723  LD      M1448  ; PB HMI COUNT Move Clean Solder
      FMOV    K0 D2032 K2
2731  END
END_PROGRAM

PROGRAM 2_MODU_C
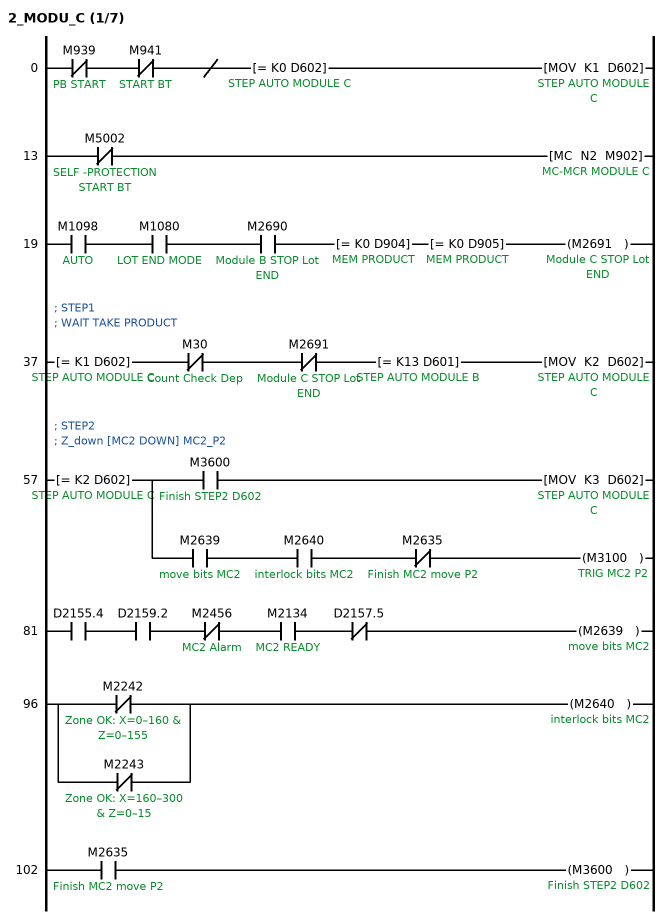
0     LDI     M939  ; PB START
      ANI     M941  ; START BT
      INV
      AND=    K0 D602  ; STEP AUTO MODULE C
      MOV     K1 D602
13    LDI     M5002  ; SELF -PROTECTION START BT
      MC      N2 M902  ; MC-MCR MODULE C
19    LD      M1098  ; AUTO
      AND     M1080  ; LOT END MODE
      AND     M2690  ; Module B STOP Lot END
      AND=    K0 D904  ; MEM PRODUCT
      AND=    K0 D905  ; MEM PRODUCT
      OUT     M2691  ; Module C STOP Lot END
; STEP1
; WAIT TAKE PRODUCT
37    LD=     K1 D602  ; STEP AUTO MODULE C
      ANI     M30  ; Count Check Dep
      ANI     M2691  ; Module C STOP Lot END
      AND=    K13 D601  ; STEP AUTO MODULE B
      MOV     K2 D602
; STEP2
; Z_down [MC2 DOWN] MC2_P2
57    LD=     K2 D602  ; STEP AUTO MODULE C
      MPS
      AND     M3600  ; Finish STEP2 D602
      MOV     K3 D602
      MPP
      AND     M2639  ; move bits MC2
      AND     M2640  ; interlock bits MC2
      ANI     M2635  ; Finish MC2 move P2
      OUT     M3100  ; TRIG MC2 P2
        [note] TRIG MC2 P2
81    LD      D2155.4
      AND     D2159.2
      ANI     M2456  ; MC2 Alarm
      AND     M2134  ; MC2 READY
      ANI     D2157.5
      OUT     M2639  ; move bits MC2
96    LDI     M2242  ; Zone OK: X=0–160 & Z=0–155
      ORI     M2243  ; Zone OK: X=160–300 & Z=0–15
      OUT     M2640  ; interlock bits MC2
102   LD      M2635  ; Finish MC2 move P2
      OUT     M3600  ; Finish STEP2 D602
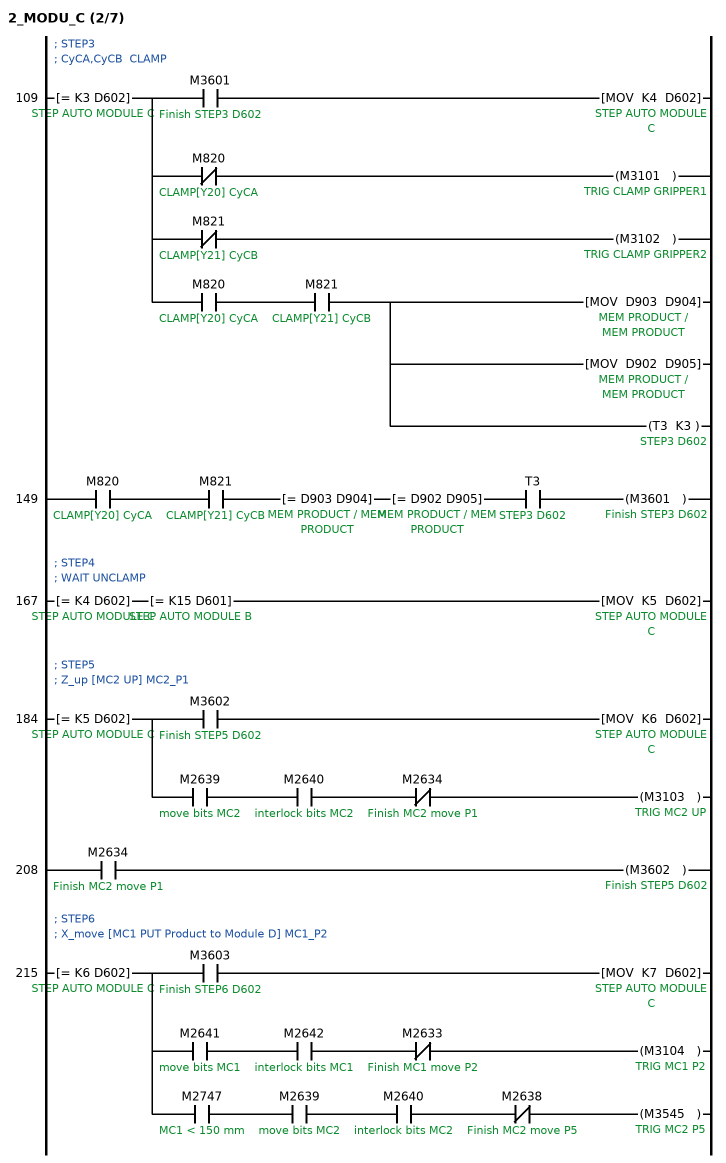
; STEP3
; CyCA,CyCB  CLAMP
109   LD=     K3 D602  ; STEP AUTO MODULE C
      MPS
      AND     M3601  ; Finish STEP3 D602
      MOV     K4 D602
      MRD
      ANI     M820  ; CLAMP[Y20] CyCA
      OUT     M3101  ; TRIG CLAMP GRIPPER1
        [note] TRIG CLAMP GRIPPER1
      MRD
      ANI     M821  ; CLAMP[Y21] CyCB
      OUT     M3102  ; TRIG CLAMP GRIPPER2
        [note] TRIG CLAMP GRIPPER2
      MPP
      AND     M820  ; CLAMP[Y20] CyCA
      AND     M821  ; CLAMP[Y21] CyCB
      MOV     D903 D904  ; MEM PRODUCT
      MOV     D902 D905  ; MEM PRODUCT
      OUT     T3 K3  ; STEP3 D602
149   LD      M820  ; CLAMP[Y20] CyCA
      AND     M821  ; CLAMP[Y21] CyCB
      AND=    D903 D904  ; MEM PRODUCT / MEM PRODUCT
      AND=    D902 D905  ; MEM PRODUCT / MEM PRODUCT
      AND     T3  ; STEP3 D602
      OUT     M3601  ; Finish STEP3 D602
; STEP4
; WAIT UNCLAMP
167   LD=     K4 D602  ; STEP AUTO MODULE C
      AND=    K15 D601  ; STEP AUTO MODULE B
      MOV     K5 D602
; STEP5
; Z_up [MC2 UP] MC2_P1
184   LD=     K5 D602  ; STEP AUTO MODULE C
      MPS
      AND     M3602  ; Finish STEP5 D602
      MOV     K6 D602
      MPP
      AND     M2639  ; move bits MC2
      AND     M2640  ; interlock bits MC2
      ANI     M2634  ; Finish MC2 move P1
      OUT     M3103  ; TRIG MC2 UP
        [note] TRIG MC2 UP
208   LD      M2634  ; Finish MC2 move P1
      OUT     M3602  ; Finish STEP5 D602
; STEP6
; X_move [MC1 PUT Product to Module D] MC1_P2
215   LD=     K6 D602  ; STEP AUTO MODULE C
      MPS
      AND     M3603  ; Finish STEP6 D602
      MOV     K7 D602
      MRD
      AND     M2641  ; move bits MC1
      AND     M2642  ; interlock bits MC1
      ANI     M2633  ; Finish MC1 move P2
      OUT     M3104  ; TRIG MC1 P2
        [note] TRIG MC1 P2
      MPP
      AND     M2747  ; MC1 < 150 mm
      AND     M2639  ; move bits MC2
      AND     M2640  ; interlock bits MC2
      ANI     M2638  ; Finish MC2 move P5
      OUT     M3545  ; TRIG MC2 P5
        [note] TRIG MC2 P5
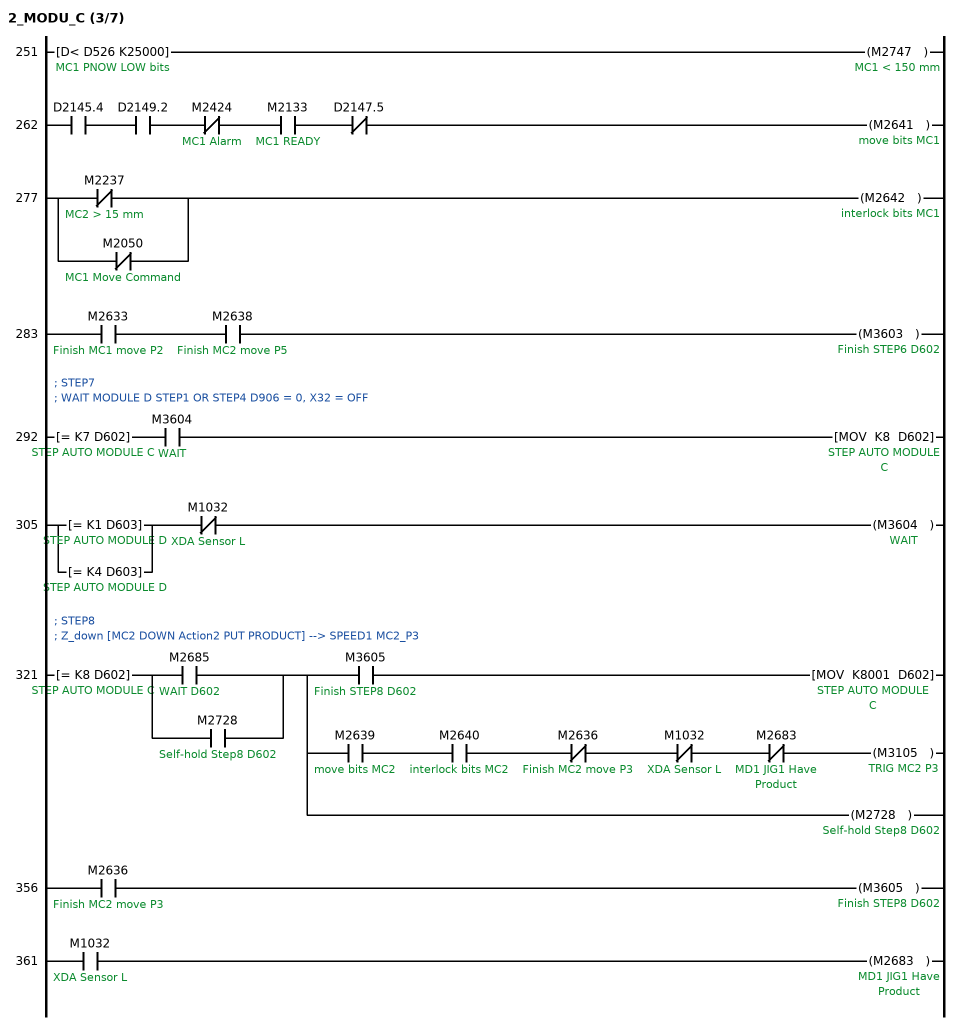
251   LDD<    D526 K25000  ; MC1 PNOW LOW bits
      OUT     M2747  ; MC1 < 150 mm
262   LD      D2145.4
      AND     D2149.2
      ANI     M2424  ; MC1 Alarm
      AND     M2133  ; MC1 READY
      ANI     D2147.5
      OUT     M2641  ; move bits MC1
277   LDI     M2237  ; MC2 > 15 mm
      ORI     M2050  ; MC1 Move Command
      OUT     M2642  ; interlock bits MC1
283   LD      M2633  ; Finish MC1 move P2
      AND     M2638  ; Finish MC2 move P5
      OUT     M3603  ; Finish STEP6 D602
; STEP7
; WAIT MODULE D STEP1 OR STEP4 D906 = 0, X32 = OFF
292   LD=     K7 D602  ; STEP AUTO MODULE C
      AND     M3604  ; WAIT
      MOV     K8 D602
305   LD=     K1 D603  ; STEP AUTO MODULE D
      OR=     K4 D603  ; STEP AUTO MODULE D
      ANI     M1032  ; XDA Sensor L
      OUT     M3604  ; WAIT
; STEP8
; Z_down [MC2 DOWN Action2 PUT PRODUCT] --> SPEED1 MC2_P3
321   LD=     K8 D602  ; STEP AUTO MODULE C
      LD      M2685  ; WAIT D602
      OR      M2728  ; Self-hold Step8 D602
      ANB
      MPS
      AND     M3605  ; Finish STEP8 D602
      MOV     K8001 D602
      MRD
      AND     M2639  ; move bits MC2
      AND     M2640  ; interlock bits MC2
      ANI     M2636  ; Finish MC2 move P3
      ANI     M1032  ; XDA Sensor L
      ANI     M2683  ; MD1 JIG1 Have Product
      OUT     M3105  ; TRIG MC2 P3
        [note] TRIG MC2 P3
      MPP
      OUT     M2728  ; Self-hold Step8 D602
356   LD      M2636  ; Finish MC2 move P3
      OUT     M3605  ; Finish STEP8 D602
361   LD      M1032  ; XDA Sensor L
      OUT     M2683  ; MD1 JIG1 Have Product
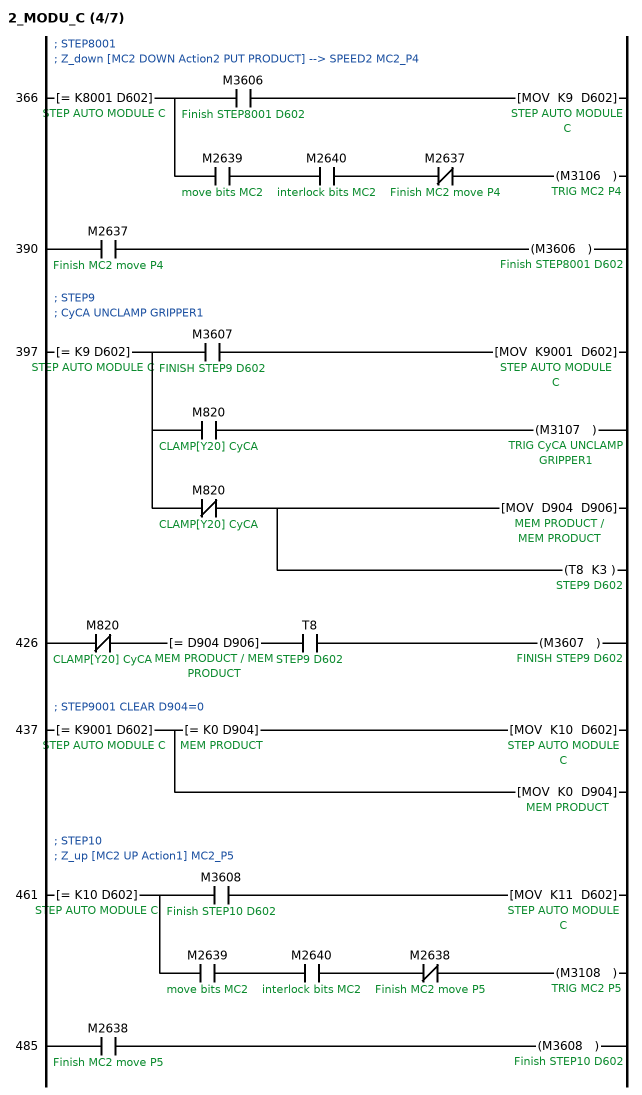
; STEP8001
; Z_down [MC2 DOWN Action2 PUT PRODUCT] --> SPEED2 MC2_P4
366   LD=     K8001 D602  ; STEP AUTO MODULE C
      MPS
      AND     M3606  ; Finish STEP8001 D602
      MOV     K9 D602
      MPP
      AND     M2639  ; move bits MC2
      AND     M2640  ; interlock bits MC2
      ANI     M2637  ; Finish MC2 move P4
      OUT     M3106  ; TRIG MC2 P4
        [note] TRIG MC2 P3
390   LD      M2637  ; Finish MC2 move P4
      OUT     M3606  ; Finish STEP8001 D602
; STEP9
; CyCA UNCLAMP GRIPPER1
397   LD=     K9 D602  ; STEP AUTO MODULE C
      MPS
      AND     M3607  ; FINISH STEP9 D602
      MOV     K9001 D602
      MRD
      AND     M820  ; CLAMP[Y20] CyCA
      OUT     M3107  ; TRIG CyCA UNCLAMP GRIPPER1
        [note] TRIG CyCA UNCLAMP GRIPPER1
      MPP
      ANI     M820  ; CLAMP[Y20] CyCA
      MOV     D904 D906  ; MEM PRODUCT
      OUT     T8 K3  ; STEP9 D602
426   LDI     M820  ; CLAMP[Y20] CyCA
      AND=    D904 D906  ; MEM PRODUCT / MEM PRODUCT
      AND     T8  ; STEP9 D602
      OUT     M3607  ; FINISH STEP9 D602
; STEP9001 CLEAR D904=0
437   LD=     K9001 D602  ; STEP AUTO MODULE C
      MPS
      AND=    K0 D904  ; MEM PRODUCT
      MOV     K10 D602
      MPP
      MOV     K0 D904
; STEP10
; Z_up [MC2 UP Action1] MC2_P5
461   LD=     K10 D602  ; STEP AUTO MODULE C
      MPS
      AND     M3608  ; Finish STEP10 D602
      MOV     K11 D602
      MPP
      AND     M2639  ; move bits MC2
      AND     M2640  ; interlock bits MC2
      ANI     M2638  ; Finish MC2 move P5
      OUT     M3108  ; TRIG MC2 P5
        [note] TRIG MC2 P5
485   LD      M2638  ; Finish MC2 move P5
      OUT     M3608  ; Finish STEP10 D602
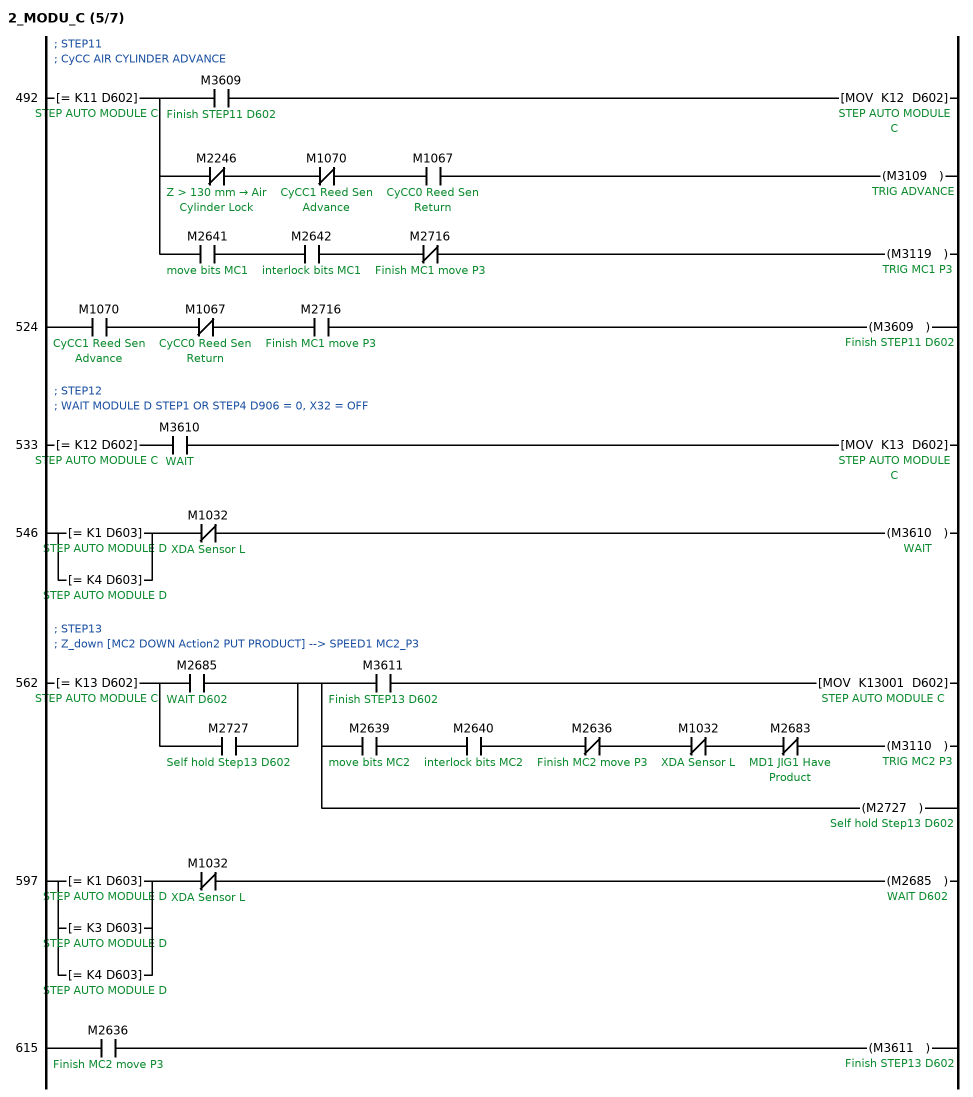
; STEP11
; CyCC AIR CYLINDER ADVANCE
492   LD=     K11 D602  ; STEP AUTO MODULE C
      MPS
      AND     M3609  ; Finish STEP11 D602
      MOV     K12 D602
      MRD
      ANI     M2246  ; Z > 130 mm → Air Cylinder Lock
      ANI     M1070  ; CyCC1 Reed Sen  Advance
      AND     M1067  ; CyCC0 Reed Sen Return
      OUT     M3109  ; TRIG ADVANCE
        [note] TRIG ADVANCE
      MPP
      AND     M2641  ; move bits MC1
      AND     M2642  ; interlock bits MC1
      ANI     M2716  ; Finish MC1 move P3
      OUT     M3119  ; TRIG MC1 P3
        [note] TRIG MC1 P3
524   LD      M1070  ; CyCC1 Reed Sen  Advance
      ANI     M1067  ; CyCC0 Reed Sen Return
      AND     M2716  ; Finish MC1 move P3
      OUT     M3609  ; Finish STEP11 D602
; STEP12
; WAIT MODULE D STEP1 OR STEP4 D906 = 0, X32 = OFF
533   LD=     K12 D602  ; STEP AUTO MODULE C
      AND     M3610  ; WAIT
      MOV     K13 D602
546   LD=     K1 D603  ; STEP AUTO MODULE D
      OR=     K4 D603  ; STEP AUTO MODULE D
      ANI     M1032  ; XDA Sensor L
      OUT     M3610  ; WAIT
; STEP13
; Z_down [MC2 DOWN Action2 PUT PRODUCT] --> SPEED1 MC2_P3
562   LD=     K13 D602  ; STEP AUTO MODULE C
      LD      M2685  ; WAIT D602
      OR      M2727  ; Self hold Step13 D602
      ANB
      MPS
      AND     M3611  ; Finish STEP13 D602
      MOV     K13001 D602
      MRD
      AND     M2639  ; move bits MC2
      AND     M2640  ; interlock bits MC2
      ANI     M2636  ; Finish MC2 move P3
      ANI     M1032  ; XDA Sensor L
      ANI     M2683  ; MD1 JIG1 Have Product
      OUT     M3110  ; TRIG MC2 P3
        [note] TRIG MC2 P3
      MPP
      OUT     M2727  ; Self hold Step13 D602
597   LD=     K1 D603  ; STEP AUTO MODULE D
      OR=     K3 D603  ; STEP AUTO MODULE D
      OR=     K4 D603  ; STEP AUTO MODULE D
      ANI     M1032  ; XDA Sensor L
      OUT     M2685  ; WAIT D602
615   LD      M2636  ; Finish MC2 move P3
      OUT     M3611  ; Finish STEP13 D602
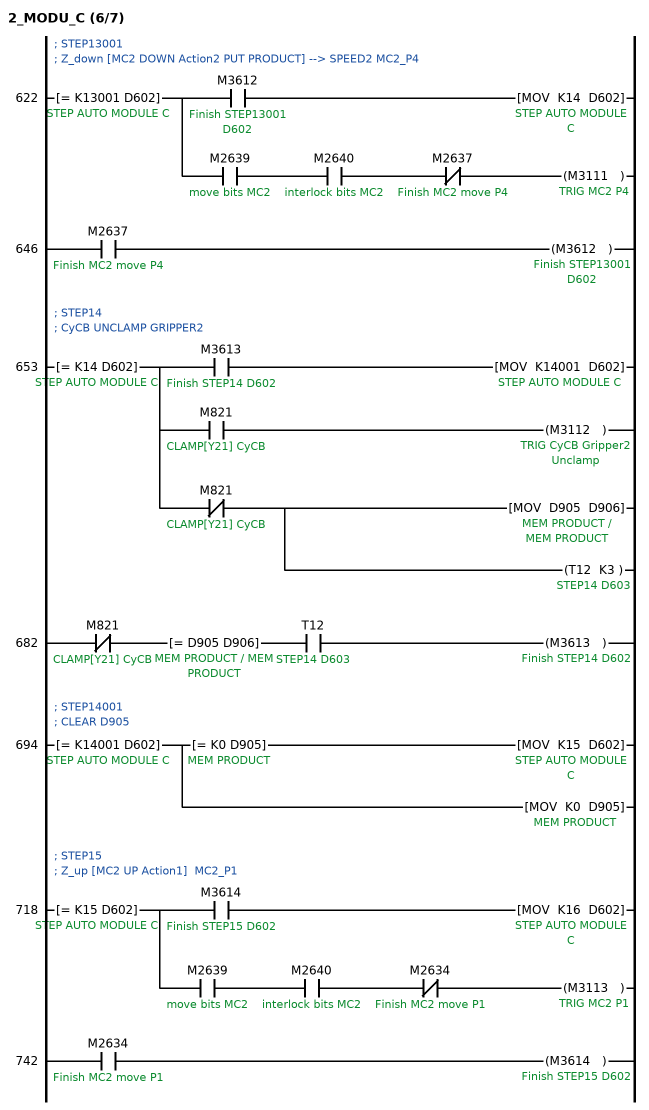
; STEP13001
; Z_down [MC2 DOWN Action2 PUT PRODUCT] --> SPEED2 MC2_P4
622   LD=     K13001 D602  ; STEP AUTO MODULE C
      MPS
      AND     M3612  ; Finish STEP13001 D602
      MOV     K14 D602
      MPP
      AND     M2639  ; move bits MC2
      AND     M2640  ; interlock bits MC2
      ANI     M2637  ; Finish MC2 move P4
      OUT     M3111  ; TRIG MC2 P4
        [note] TRIG MC2 P4
646   LD      M2637  ; Finish MC2 move P4
      OUT     M3612  ; Finish STEP13001 D602
; STEP14
; CyCB UNCLAMP GRIPPER2
653   LD=     K14 D602  ; STEP AUTO MODULE C
      MPS
      AND     M3613  ; Finish STEP14 D602
      MOV     K14001 D602
      MRD
      AND     M821  ; CLAMP[Y21] CyCB
      OUT     M3112  ; TRIG CyCB Gripper2 Unclamp
        [note] TRIG CyCB Gripper2 Unclamp
      MPP
      ANI     M821  ; CLAMP[Y21] CyCB
      MOV     D905 D906
      OUT     T12 K3  ; STEP14 D603
682   LDI     M821  ; CLAMP[Y21] CyCB
      AND=    D905 D906  ; MEM PRODUCT / MEM PRODUCT
      AND     T12  ; STEP14 D603
      OUT     M3613  ; Finish STEP14 D602
; STEP14001
; CLEAR D905
694   LD=     K14001 D602  ; STEP AUTO MODULE C
      MPS
      AND=    K0 D905  ; MEM PRODUCT
      MOV     K15 D602
      MPP
      MOV     K0 D905
; STEP15
; Z_up [MC2 UP Action1]  MC2_P1
718   LD=     K15 D602  ; STEP AUTO MODULE C
      MPS
      AND     M3614  ; Finish STEP15 D602
      MOV     K16 D602
      MPP
      AND     M2639  ; move bits MC2
      AND     M2640  ; interlock bits MC2
      ANI     M2634  ; Finish MC2 move P1
      OUT     M3113  ; TRIG MC2 P1
        [note] TRIG MC2 P1
742   LD      M2634  ; Finish MC2 move P1
      OUT     M3614  ; Finish STEP15 D602
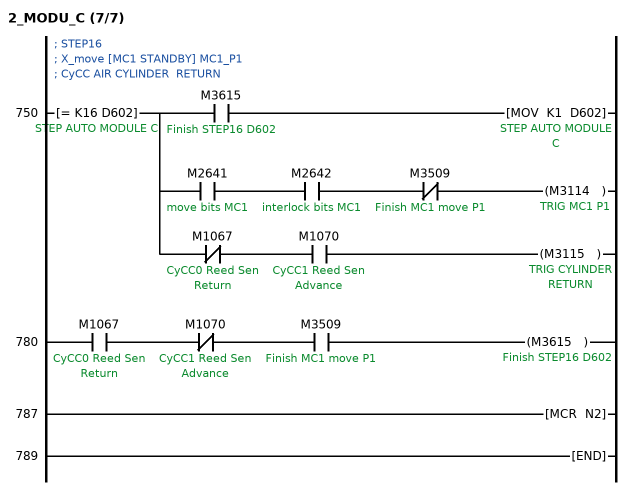
; STEP16
; X_move [MC1 STANDBY] MC1_P1
; CyCC AIR CYLINDER  RETURN
750   LD=     K16 D602  ; STEP AUTO MODULE C
      MPS
      AND     M3615  ; Finish STEP16 D602
      MOV     K1 D602
      MRD
      AND     M2641  ; move bits MC1
      AND     M2642  ; interlock bits MC1
      ANI     M3509  ; Finish MC1 move P1
      OUT     M3114  ; TRIG MC1 P1
        [note] TRIG MC1 P1
      MPP
      ANI     M1067  ; CyCC0 Reed Sen Return
      AND     M1070  ; CyCC1 Reed Sen  Advance
      OUT     M3115  ; TRIG CYLINDER RETURN
        [note] TRIG CYLINDER RETURN
780   LD      M1067  ; CyCC0 Reed Sen Return
      ANI     M1070  ; CyCC1 Reed Sen  Advance
      AND     M3509  ; Finish MC1 move P1
      OUT     M3615  ; Finish STEP16 D602
787   MCR     N2
789   END
END_PROGRAM

PROGRAM 3_MODU_D
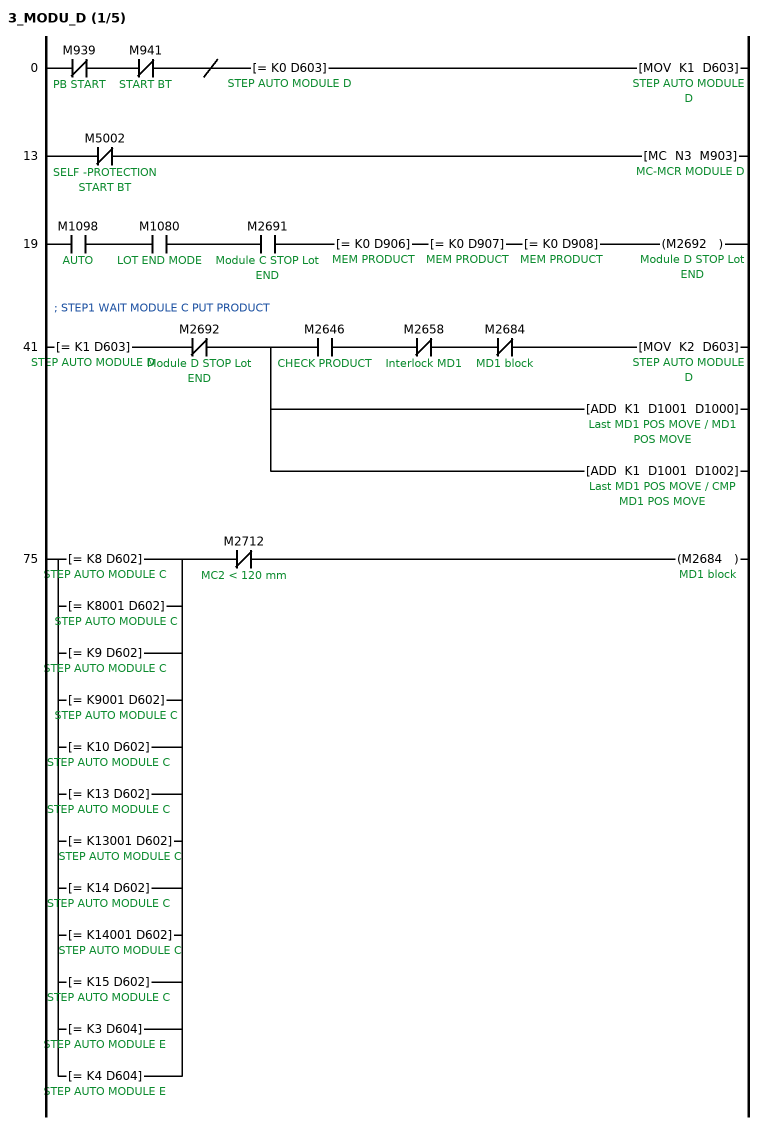
0     LDI     M939  ; PB START
      ANI     M941  ; START BT
      INV
      AND=    K0 D603  ; STEP AUTO MODULE D
      MOV     K1 D603
13    LDI     M5002  ; SELF -PROTECTION START BT
      MC      N3 M903  ; MC-MCR MODULE D
19    LD      M1098  ; AUTO
      AND     M1080  ; LOT END MODE
      AND     M2691  ; Module C STOP Lot END
      AND=    K0 D906  ; MEM PRODUCT
      AND=    K0 D907  ; MEM PRODUCT
      AND=    K0 D908  ; MEM PRODUCT
      OUT     M2692  ; Module D STOP Lot END
; STEP1 WAIT MODULE C PUT PRODUCT
41    LD=     K1 D603  ; STEP AUTO MODULE D
      ANI     M2692  ; Module D STOP Lot END
      MPS
      AND     M2646  ; CHECK PRODUCT
      ANI     M2658  ; Interlock MD1
      ANI     M2684  ; MD1 block
      MOV     K2 D603
      MPP
      ADD     K1 D1001 D1000  ; Last MD1 POS MOVE / MD1 POS MOVE
      ADD     K1 D1001 D1002  ; CMP MD1 POS MOVE
75    LD=     K8 D602  ; STEP AUTO MODULE C
      OR=     K8001 D602  ; STEP AUTO MODULE C
      OR=     K9 D602  ; STEP AUTO MODULE C
      OR=     K9001 D602  ; STEP AUTO MODULE C
      OR=     K10 D602  ; STEP AUTO MODULE C
      OR=     K13 D602  ; STEP AUTO MODULE C
      OR=     K13001 D602  ; STEP AUTO MODULE C
      OR=     K14 D602  ; STEP AUTO MODULE C
      OR=     K14001 D602  ; STEP AUTO MODULE C
      OR=     K15 D602  ; STEP AUTO MODULE C
      OR=     K3 D604  ; STEP AUTO MODULE E
      OR=     K4 D604  ; STEP AUTO MODULE E
      ANI     M2712  ; MC2 < 120 mm
      OUT     M2684  ; MD1 block
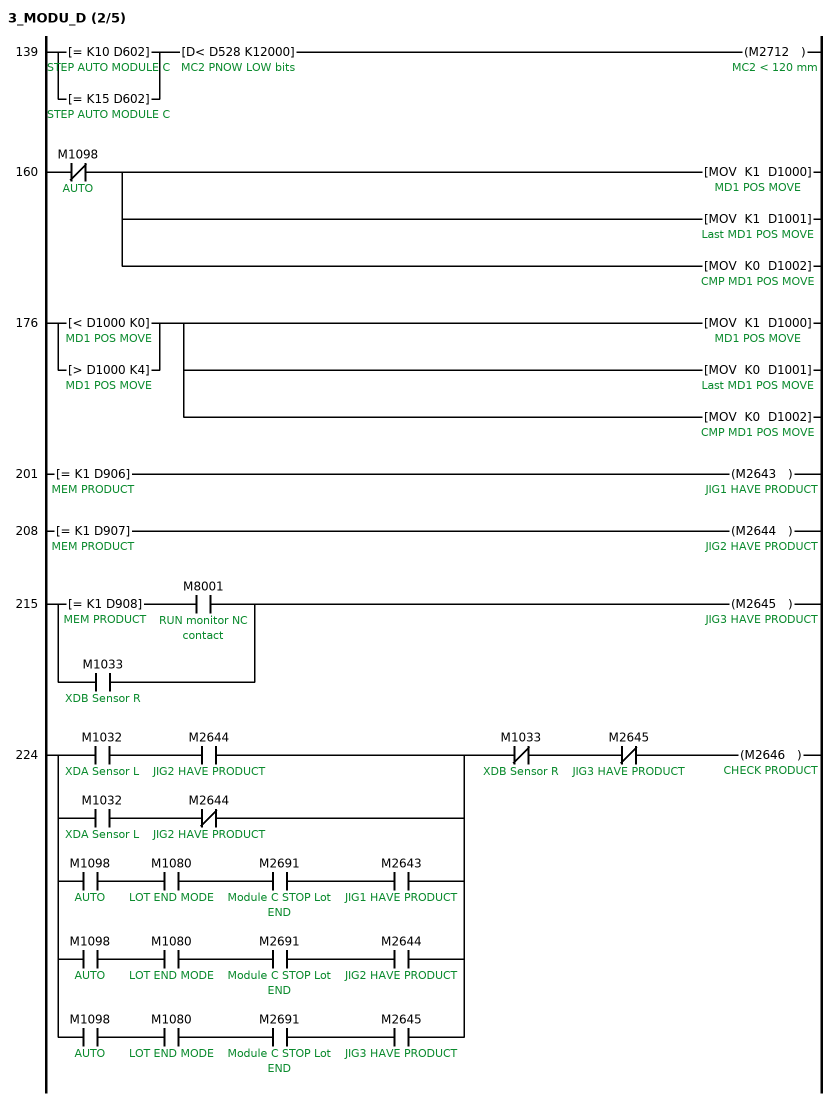
139   LD=     K10 D602  ; STEP AUTO MODULE C
      OR=     K15 D602  ; STEP AUTO MODULE C
      ANDD<   D528 K12000  ; MC2 PNOW LOW bits
      OUT     M2712  ; MC2 < 120 mm
160   LDI     M1098  ; AUTO
      MOV     K1 D1000
      MOV     K1 D1001
      MOV     K0 D1002
176   LD<     D1000 K0  ; MD1 POS MOVE
      OR>     D1000 K4  ; MD1 POS MOVE
      MOV     K1 D1000
      MOV     K0 D1001
      MOV     K0 D1002
201   LD=     K1 D906  ; MEM PRODUCT
      OUT     M2643  ; JIG1 HAVE PRODUCT
208   LD=     K1 D907  ; MEM PRODUCT
      OUT     M2644  ; JIG2 HAVE PRODUCT
215   LD=     K1 D908  ; MEM PRODUCT
      AND     M8001  ; RUN monitor NC contact
      OR      M1033  ; XDB Sensor R
      OUT     M2645  ; JIG3 HAVE PRODUCT
224   LD      M1032  ; XDA Sensor L
      AND     M2644  ; JIG2 HAVE PRODUCT
      LD      M1032  ; XDA Sensor L
      ANI     M2644  ; JIG2 HAVE PRODUCT
      ORB
      LD      M1098  ; AUTO
      AND     M1080  ; LOT END MODE
      AND     M2691  ; Module C STOP Lot END
      AND     M2643  ; JIG1 HAVE PRODUCT
      ORB
      LD      M1098  ; AUTO
      AND     M1080  ; LOT END MODE
      AND     M2691  ; Module C STOP Lot END
      AND     M2644  ; JIG2 HAVE PRODUCT
      ORB
      LD      M1098  ; AUTO
      AND     M1080  ; LOT END MODE
      AND     M2691  ; Module C STOP Lot END
      AND     M2645  ; JIG3 HAVE PRODUCT
      ORB
      ANI     M1033  ; XDB Sensor R
      ANI     M2645  ; JIG3 HAVE PRODUCT
      OUT     M2646  ; CHECK PRODUCT
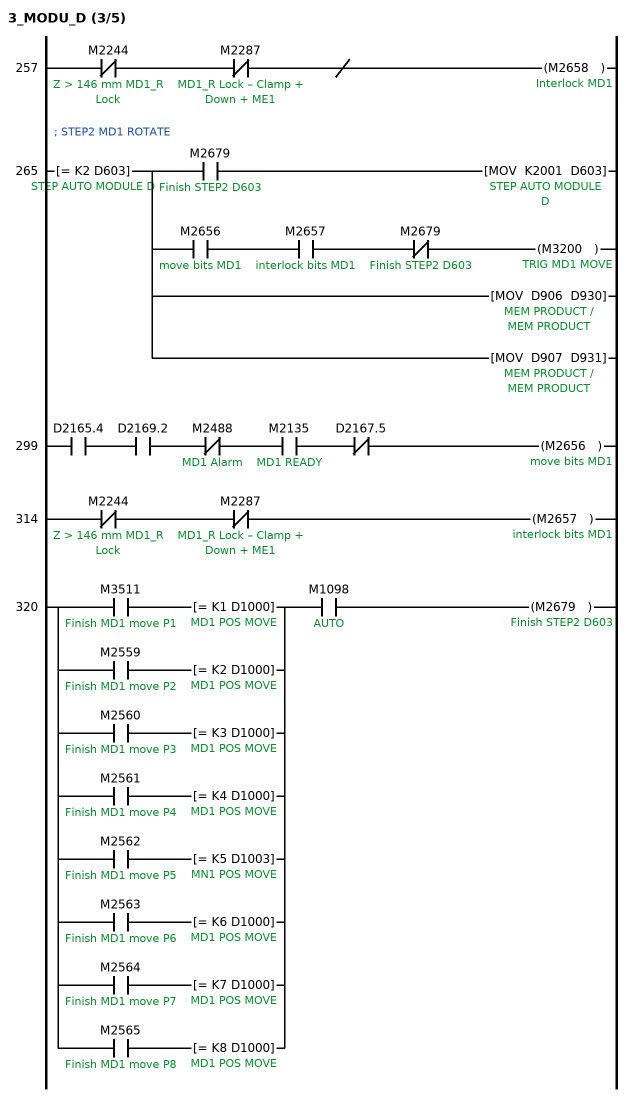
257   LDI     M2244  ; Z > 146 mm MD1_R Lock
      ANI     M2287  ; MD1_R Lock – Clamp + Down + ME1
      INV
      OUT     M2658  ; Interlock MD1
; STEP2 MD1 ROTATE
265   LD=     K2 D603  ; STEP AUTO MODULE D
      MPS
      AND     M2679  ; Finish STEP2 D603
      MOV     K2001 D603
      MRD
      AND     M2656  ; move bits MD1
      AND     M2657  ; interlock bits MD1
      ANI     M2679  ; Finish STEP2 D603
      OUT     M3200  ; TRIG MD1 MOVE
        [note] TRIG MD1 MOVE
      MPP
      MOV     D906 D930  ; MEM PRODUCT
      MOV     D907 D931  ; MEM PRODUCT
299   LD      D2165.4
      AND     D2169.2
      ANI     M2488  ; MD1 Alarm
      AND     M2135  ; MD1 READY
      ANI     D2167.5
      OUT     M2656  ; move bits MD1
314   LDI     M2244  ; Z > 146 mm MD1_R Lock
      ANI     M2287  ; MD1_R Lock – Clamp + Down + ME1
      OUT     M2657  ; interlock bits MD1
320   LD      M3511  ; Finish MD1 move P1
      AND=    K1 D1000  ; MD1 POS MOVE
      LD      M2559  ; Finish MD1 move P2
      AND=    K2 D1000  ; MD1 POS MOVE
      ORB
      LD      M2560  ; Finish MD1 move P3
      AND=    K3 D1000  ; MD1 POS MOVE
      ORB
      LD      M2561  ; Finish MD1 move P4
      AND=    K4 D1000  ; MD1 POS MOVE
      ORB
      LD      M2562  ; Finish MD1 move P5
      AND=    K5 D1003  ; MN1 POS MOVE
      ORB
      LD      M2563  ; Finish MD1 move P6
      AND=    K6 D1000  ; MD1 POS MOVE
      ORB
      LD      M2564  ; Finish MD1 move P7
      AND=    K7 D1000  ; MD1 POS MOVE
      ORB
      LD      M2565  ; Finish MD1 move P8
      AND=    K8 D1000  ; MD1 POS MOVE
      ORB
      AND     M1098  ; AUTO
      OUT     M2679  ; Finish STEP2 D603
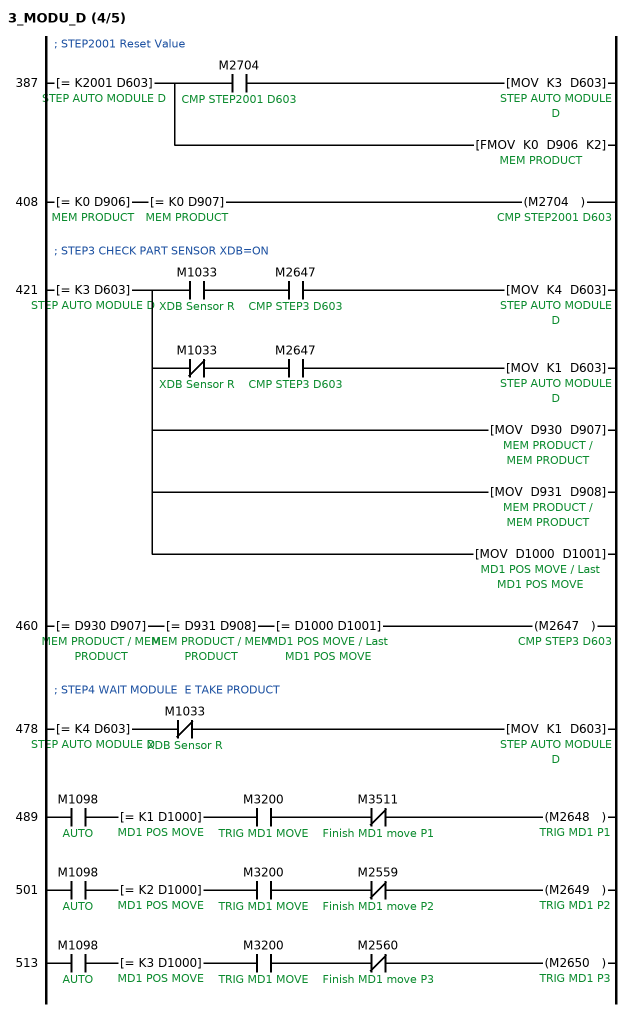
; STEP2001 Reset Value
387   LD=     K2001 D603  ; STEP AUTO MODULE D
      MPS
      AND     M2704  ; CMP STEP2001 D603
      MOV     K3 D603
      MPP
      FMOV    K0 D906 K2
408   LD=     K0 D906  ; MEM PRODUCT
      AND=    K0 D907  ; MEM PRODUCT
      OUT     M2704  ; CMP STEP2001 D603
; STEP3 CHECK PART SENSOR XDB=ON
421   LD=     K3 D603  ; STEP AUTO MODULE D
      MPS
      AND     M1033  ; XDB Sensor R
      AND     M2647  ; CMP STEP3 D603
      MOV     K4 D603
      MRD
      ANI     M1033  ; XDB Sensor R
      AND     M2647  ; CMP STEP3 D603
      MOV     K1 D603
      MPP
      MOV     D930 D907
      MOV     D931 D908
      MOV     D1000 D1001
460   LD=     D930 D907  ; MEM PRODUCT / MEM PRODUCT
      AND=    D931 D908  ; MEM PRODUCT / MEM PRODUCT
      AND=    D1000 D1001  ; MD1 POS MOVE / Last MD1 POS MOVE
      OUT     M2647  ; CMP STEP3 D603
; STEP4 WAIT MODULE  E TAKE PRODUCT
478   LD=     K4 D603  ; STEP AUTO MODULE D
      ANI     M1033  ; XDB Sensor R
      MOV     K1 D603
489   LD      M1098  ; AUTO
      AND=    K1 D1000  ; MD1 POS MOVE
      AND     M3200  ; TRIG MD1 MOVE
      ANI     M3511  ; Finish MD1 move P1
      OUT     M2648  ; TRIG MD1 P1
501   LD      M1098  ; AUTO
      AND=    K2 D1000  ; MD1 POS MOVE
      AND     M3200  ; TRIG MD1 MOVE
      ANI     M2559  ; Finish MD1 move P2
      OUT     M2649  ; TRIG MD1 P2
513   LD      M1098  ; AUTO
      AND=    K3 D1000  ; MD1 POS MOVE
      AND     M3200  ; TRIG MD1 MOVE
      ANI     M2560  ; Finish MD1 move P3
      OUT     M2650  ; TRIG MD1 P3
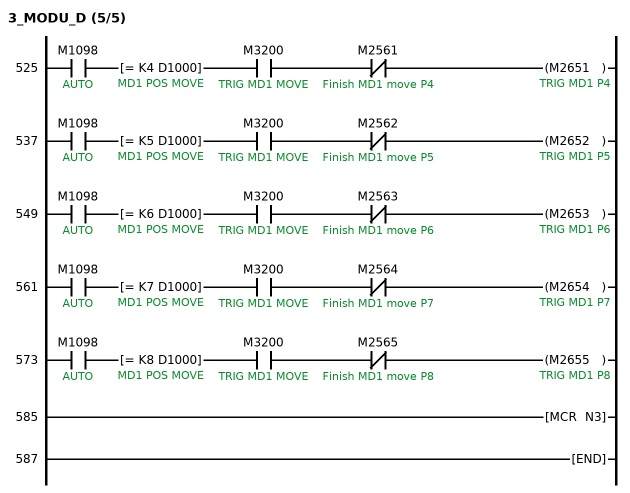
525   LD      M1098  ; AUTO
      AND=    K4 D1000  ; MD1 POS MOVE
      AND     M3200  ; TRIG MD1 MOVE
      ANI     M2561  ; Finish MD1 move P4
      OUT     M2651  ; TRIG MD1 P4
537   LD      M1098  ; AUTO
      AND=    K5 D1000  ; MD1 POS MOVE
      AND     M3200  ; TRIG MD1 MOVE
      ANI     M2562  ; Finish MD1 move P5
      OUT     M2652  ; TRIG MD1 P5
549   LD      M1098  ; AUTO
      AND=    K6 D1000  ; MD1 POS MOVE
      AND     M3200  ; TRIG MD1 MOVE
      ANI     M2563  ; Finish MD1 move P6
      OUT     M2653  ; TRIG MD1 P6
561   LD      M1098  ; AUTO
      AND=    K7 D1000  ; MD1 POS MOVE
      AND     M3200  ; TRIG MD1 MOVE
      ANI     M2564  ; Finish MD1 move P7
      OUT     M2654  ; TRIG MD1 P7
573   LD      M1098  ; AUTO
      AND=    K8 D1000  ; MD1 POS MOVE
      AND     M3200  ; TRIG MD1 MOVE
      ANI     M2565  ; Finish MD1 move P8
      OUT     M2655  ; TRIG MD1 P8
585   MCR     N3
587   END
END_PROGRAM

PROGRAM 4_MODU_E
